RoboDK station: kr30 cnc 072119 second half.rdk

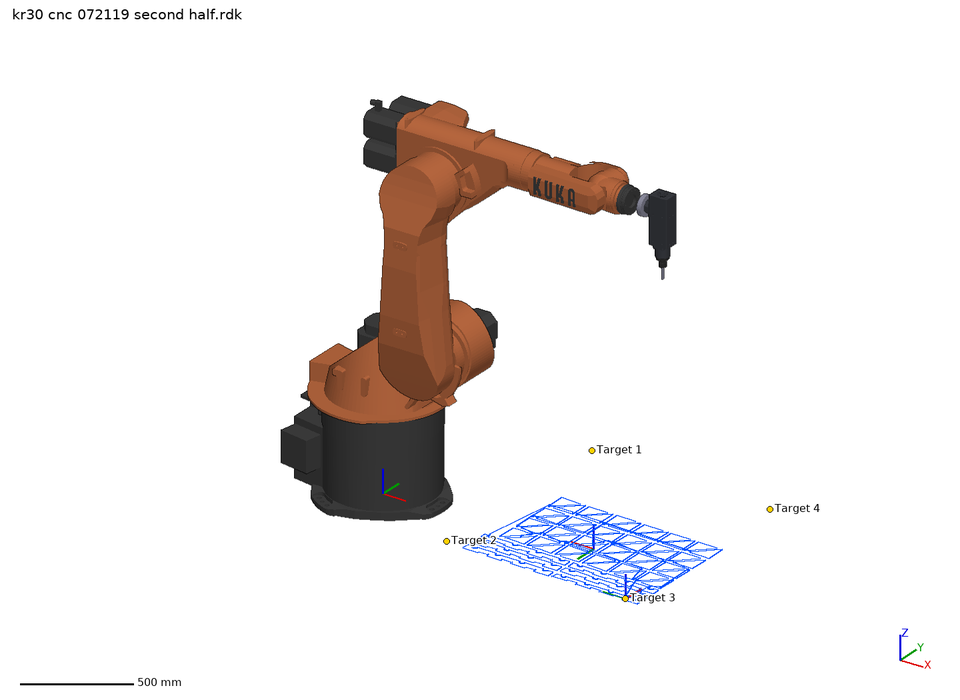
[picture v0: the station drawn from its stored meshes, robots at their saved joint values, targets as dots, program paths as lines]
Station kr30 cnc 072119 second half. Poses are relative to the parent item; angles as X-Y-Z fixed-axis rotations.
  - frame GIGASHEEN Base at (0, 0, 0) mm
    - robot GIGASHEEN (model KUKA KR 30 HA): 6 axes, payload 30 kg, reach 2033 mm, repeatability 0.05 mm, weight 665 kg
        modified DH rows (alpha deg, a mm, theta deg, d mm): 0, 0, 0, 815; -90, 350, 0, 0; 0, 850, -90, 0; -90, 145, 0, 820; 90, 0, 0, 0; -90, 0, 180, 170
        joint limits [-185, -135, -120, -350, -119, -350] to [185, 35, 158, 350, 119, 350]; home [0, -90, 90, 0, 0, 0]; saved at [0, -90, 90, 0, 0, 0]
      - tool 1/2" End Mill TCP, TCP at (337.71, -2.2, 160.57) mm, rotated rx 0 ry 90 rz 0 deg, size 415.8 x 102 x 153.6 mm
    - target Target 1 (joint target) at (982.46, 202.21, 406.25) mm, rotated rx -179.95 ry 0.15 rz -89.48 deg; joints [7.49, -59.642, 144.935, 97.969, -90.801, -4.608] of GIGASHEEN
    - target Target 2 (joint target) at (986.83, -921.64, 412.07) mm, rotated rx -179.94 ry 0.15 rz -89.48 deg; joints [51.766, -38.608, 94.384, 136.851, -116.554, -22.567] of GIGASHEEN
    - target Target 3 (joint target) at (1949.02, -919.97, 396.91) mm, rotated rx -179.94 ry 0.14 rz 179.61 deg; joints [29.5, -22.76, 62.288, 41.088, -47.759, -30.404] of GIGASHEEN
    - target Target 4 (joint target) at (1949.02, 190.94, 391.63) mm, rotated rx -179.94 ry 0.14 rz 179.61 deg; joints [-6.898, -35.989, 90.741, -8.88, -55.221, 5.167] of GIGASHEEN
  - machining project Machining Settings: C:/Users/liqui/OneDrive/Desktop/second half pipe jig.apt | rotZ(0) | rotX(0)*rotY(0) | rotZ(0)
  - program Prog2 (4 instructions, listed below)
  - frame Table at (1949.02, -919.97, 396.91) mm, rotated rx 0.87 ry 0.27 rz 90 deg
    - frame Frame 4 at (440, 480, -70) mm, rotated rx 0 ry 0 rz 90 deg
  - program Machining (1046 instructions, listed below)
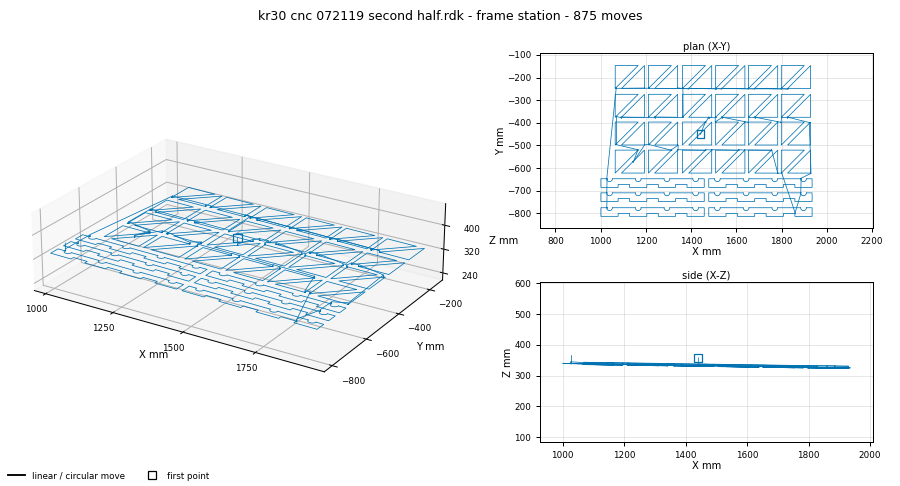
[picture p0: tool path of kr30 cnc 072119 second half.rdk in frame station, 875 of 879 moves have a stored position in this frame; points joined in program order, loops and branches not executed]

--- program Prog2 (robot GIGASHEEN) ---
  MoveJ (plywood back right safe) [its target is no longer in the station]
  MoveL (plywood back left safe) [its target is no longer in the station]
  MoveL (plywood front left safe) [its target is no longer in the station]
  MoveL (plywood front right safe) [its target is no longer in the station]

--- program Machining (robot GIGASHEEN) ---
  Smooth(1)
  Set Ref.: Frame 4
  Set Tool: 1/2" End Mill TCP
  Show 1/2" End Mill TCP
  Print: /'1001'
  Print: /''
  Print: /'2D Contour8'
  Set speed (500.0 mm/s)
  MoveJ 1 to (26.81, -31, 25) mm, rotated rx 180 ry 0 rz 0 deg; joints [21.751, -50.614, 128.61, 22.256, -77.995, -4.246]
  MoveL 2 to (26.81, -31, 25) mm, rotated rx 180 ry 0 rz 0 deg; joints [21.751, -50.614, 128.61, 22.256, -77.995, -4.246]
  MoveL 3 to (26.81, -31, 15) mm, rotated rx -180 ry 0 rz 0 deg; joints [21.756, -49.905, 128.509, 22.213, -78.558, -4.012]
  MoveL 4 to (26.81, -31, 15) mm, rotated rx -180 ry 0 rz 0 deg; joints [21.756, -49.905, 128.509, 22.213, -78.558, -4.012]
  Set speed (500.0 mm/s)
  MoveL 5 to (26.81, -31, 5) mm, rotated rx -180 ry 0 rz 0 deg; joints [21.761, -49.194, 128.4, 22.173, -79.115, -3.781]
  Set speed (25.4 mm/s)
  MoveL 6 to (26.81, -31, 1) mm, rotated rx -180 ry 0 rz 0 deg; joints [21.762, -48.909, 128.353, 22.158, -79.337, -3.69]
  MoveL 7 to (26.81, -31, -0.37) mm, rotated rx -180 ry 0 rz 0 deg; joints [21.763, -48.811, 128.337, 22.153, -79.412, -3.659]
  MoveC 8 to (26.94, -31.13, -0.81) mm, rotated rx -180 ry 0 rz 0 deg; joints [21.76, -48.784, 128.345, 22.147, -79.444, -3.645] to (27.26, -31.45, -1) mm, rotated rx 180 ry 0 rz 0 deg; joints [21.751, -48.782, 128.375, 22.136, -79.474, -3.631]
  Set speed (50.8 mm/s)
  MoveL 9 to (27.71, -31.9, -1) mm, rotated rx -180 ry 0 rz 0 deg; joints [21.739, -48.798, 128.421, 22.122, -79.5, -3.618]
  MoveC 10 to (27.89, -32.35, -1) mm, rotated rx -180 ry 0 rz 0 deg; joints [21.723, -48.807, 128.447, 22.104, -79.515, -3.608] to (27.71, -32.8, -1) mm, rotated rx -180 ry 0 rz 0 deg; joints [21.7, -48.806, 128.447, 22.081, -79.514, -3.604]
  MoveL 11 to (-23.07, -83.55, -1) mm, rotated rx 180 ry 0 rz 0 deg; joints [18.628, -47.91, 126.057, 19.06, -77.908, -3.574]
  MoveL 12 to (-23.07, 17.99, -1) mm, rotated rx 180 ry 0 rz 0 deg; joints [22.986, -46.905, 123.177, 23.67, -76.514, -5.195]
  MoveL 13 to (78.53, 17.99, -1) mm, rotated rx -180 ry 0 rz 0 deg; joints [24.923, -49.575, 130.527, 25.253, -80.933, -3.575]
  MoveL 14 to (27.71, -32.8, -1) mm, rotated rx -180 ry 0 rz 0 deg; joints [21.7, -48.806, 128.447, 22.081, -79.514, -3.604]
  MoveC 15 to (27.26, -32.98, -1) mm, rotated rx -180 ry 0 rz 0 deg; joints [21.683, -48.796, 128.419, 22.065, -79.497, -3.608] to (26.81, -32.8, -1) mm, rotated rx -180 ry 0 rz 0 deg; joints [21.684, -48.783, 128.381, 22.067, -79.474, -3.618]
  MoveL 16 to (26.36, -32.35, -1) mm, rotated rx -180 ry 0 rz 0 deg; joints [21.696, -48.767, 128.335, 22.082, -79.447, -3.631]
  MoveC 17 to (26.04, -32.03, -0.81) mm, rotated rx -180 ry 0 rz 0 deg; joints [21.704, -48.769, 128.305, 22.092, -79.418, -3.645] to (25.91, -31.9, -0.37) mm, rotated rx -180 ry 0 rz 0 deg; joints [21.707, -48.796, 128.297, 22.098, -79.385, -3.659]
  Set speed (500.0 mm/s)
  MoveL 18 to (25.91, -31.9, 5) mm, rotated rx -180 ry 0 rz 0 deg; joints [21.705, -49.179, 128.36, 22.119, -79.089, -3.781]
  MoveL 19 to (4.1, -85.45, 5) mm, rotated rx 180 ry 0 rz 0 deg; joints [18.952, -49.087, 128.208, 19.324, -78.85, -3.309]
  Set speed (25.4 mm/s)
  MoveL 20 to (4.1, -85.45, 1) mm, rotated rx -180 ry 0 rz 0 deg; joints [18.954, -48.802, 128.162, 19.311, -79.074, -3.229]
  MoveL 21 to (4.1, -85.45, -0.37) mm, rotated rx -180 ry 0 rz 0 deg; joints [18.954, -48.705, 128.146, 19.306, -79.151, -3.202]
  MoveC 22 to (4.1, -85.27, -0.81) mm, rotated rx -180 ry 0 rz 0 deg; joints [18.963, -48.672, 128.135, 19.314, -79.173, -3.195] to (4.1, -84.82, -1) mm, rotated rx 180 ry 0 rz 0 deg; joints [18.983, -48.655, 128.122, 19.334, -79.178, -3.198]
  Set speed (50.8 mm/s)
  MoveL 23 to (4.1, -84.18, -1) mm, rotated rx 180 ry 0 rz 0 deg; joints [19.012, -48.649, 128.106, 19.364, -79.169, -3.206]
  MoveC 24 to (4.29, -83.73, -1) mm, rotated rx 180 ry 0 rz 0 deg; joints [19.035, -48.65, 128.108, 19.387, -79.172, -3.21] to (4.74, -83.55, -1) mm, rotated rx 180 ry 0 rz 0 deg; joints [19.05, -48.661, 128.137, 19.402, -79.19, -3.207]
  MoveL 25 to (106.34, -83.55, -1) mm, rotated rx -180 ry 0 rz 0 deg; joints [20.764, -51.132, 135.495, 20.883, -83.861, -1.734]
  MoveL 26 to (106.34, 17.99, -1) mm, rotated rx -180 ry 0 rz 0 deg; joints [25.508, -50.235, 132.469, 25.761, -82.126, -3.095]
  MoveL 27 to (4.74, -83.55, -1) mm, rotated rx 180 ry 0 rz 0 deg; joints [19.05, -48.661, 128.137, 19.402, -79.19, -3.207]
  MoveC 28 to (4.29, -83.73, -1) mm, rotated rx -180 ry 0 rz 0 deg; joints [19.035, -48.65, 128.108, 19.387, -79.172, -3.21] to (3.84, -83.55, -1) mm, rotated rx 180 ry 0 rz 0 deg; joints [19.036, -48.637, 128.07, 19.39, -79.149, -3.219]
  MoveL 29 to (3.39, -83.1, -1) mm, rotated rx 180 ry 0 rz 0 deg; joints [19.05, -48.621, 128.025, 19.405, -79.122, -3.231]
  MoveC 30 to (3.07, -82.78, -0.81) mm, rotated rx -180 ry 0 rz 0 deg; joints [19.059, -48.623, 127.996, 19.417, -79.093, -3.243] to (2.94, -82.65, -0.37) mm, rotated rx -180 ry 0 rz 0 deg; joints [19.062, -48.651, 127.988, 19.423, -79.06, -3.256]
  Set speed (500.0 mm/s)
  MoveL 31 to (2.94, -82.65, 5) mm, rotated rx 180 ry 0 rz 0 deg; joints [19.06, -49.031, 128.05, 19.441, -78.76, -3.363]
  MoveL 32 to (-7.94, -102.8, 5) mm, rotated rx -180 ry 0 rz 0 deg; joints [17.99, -48.905, 127.74, 18.364, -78.518, -3.226]
  Set speed (25.4 mm/s)
  MoveL 33 to (-7.94, -102.8, 1) mm, rotated rx -180 ry 0 rz 0 deg; joints [17.992, -48.623, 127.693, 18.351, -78.743, -3.15]
  MoveL 34 to (-7.94, -102.8, -0.37) mm, rotated rx -180 ry 0 rz 0 deg; joints [17.992, -48.526, 127.677, 18.346, -78.819, -3.124]
  MoveC 35 to (-7.94, -102.98, -0.81) mm, rotated rx -180 ry 0 rz 0 deg; joints [17.984, -48.496, 127.676, 18.336, -78.847, -3.114] to (-7.94, -103.43, -1) mm, rotated rx 180 ry 0 rz 0 deg; joints [17.964, -48.486, 127.685, 18.314, -78.863, -3.104]
  Set speed (50.8 mm/s)
  MoveL 36 to (-7.94, -104.07, -1) mm, rotated rx 180 ry 0 rz 0 deg; joints [17.935, -48.491, 127.7, 18.285, -78.871, -3.096]
  MoveC 37 to (-8.13, -104.52, -1) mm, rotated rx 180 ry 0 rz 0 deg; joints [17.912, -48.49, 127.697, 18.261, -78.868, -3.092] to (-8.57, -104.7, -1) mm, rotated rx -180 ry 0 rz 0 deg; joints [17.897, -48.479, 127.668, 18.247, -78.849, -3.095]
  MoveL 38 to (-23.07, -104.7, -1) mm, rotated rx -180 ry 0 rz 0 deg; joints [17.689, -48.086, 126.578, 18.079, -78.174, -3.278]
  MoveL 39 to (-23.07, -206.24, -1) mm, rotated rx -180 ry 0 rz 0 deg; joints [13.051, -48.78, 128.687, 13.281, -79.301, -2.035]
  MoveL 40 to (78.53, -104.7, -1) mm, rotated rx 180 ry 0 rz 0 deg; joints [19.258, -50.66, 134.059, 19.406, -82.901, -1.917]
  MoveL 41 to (-8.57, -104.7, -1) mm, rotated rx -180 ry 0 rz 0 deg; joints [17.897, -48.479, 127.668, 18.247, -78.849, -3.095]
  MoveC 42 to (-9.02, -104.52, -1) mm, rotated rx -180 ry 0 rz 0 deg; joints [17.899, -48.466, 127.63, 18.251, -78.826, -3.103] to (-9.21, -104.07, -1) mm, rotated rx -180 ry 0 rz 0 deg; joints [17.917, -48.457, 127.605, 18.27, -78.812, -3.112]
  MoveL 43 to (-9.21, -103.43, -1) mm, rotated rx -180 ry 0 rz 0 deg; joints [17.945, -48.452, 127.59, 18.299, -78.804, -3.12]
  MoveC 44 to (-9.21, -102.98, -0.81) mm, rotated rx -180 ry 0 rz 0 deg; joints [17.965, -48.462, 127.581, 18.321, -78.788, -3.13] to (-9.21, -102.8, -0.37) mm, rotated rx 180 ry 0 rz 0 deg; joints [17.974, -48.492, 127.582, 18.331, -78.76, -3.141]
  Set speed (500.0 mm/s)
  MoveL 45 to (-9.21, -102.8, 5) mm, rotated rx -180 ry 0 rz 0 deg; joints [17.971, -48.871, 127.644, 18.349, -78.46, -3.242]
  MoveL 46 to (-41.36, -102.91, 5) mm, rotated rx -180 ry 0 rz 0 deg; joints [17.509, -47.974, 125.216, 17.98, -76.975, -3.637]
  Set speed (25.4 mm/s)
  MoveL 47 to (-41.36, -102.91, 1) mm, rotated rx -180 ry 0 rz 0 deg; joints [17.511, -47.7, 125.171, 17.966, -77.192, -3.565]
  MoveL 48 to (-41.36, -102.91, -0.36) mm, rotated rx -180 ry 0 rz 0 deg; joints [17.511, -47.607, 125.155, 17.961, -77.266, -3.541]
  MoveC 49 to (-41.23, -103.04, -0.81) mm, rotated rx -180 ry 0 rz 0 deg; joints [17.507, -47.581, 125.163, 17.955, -77.298, -3.529] to (-40.91, -103.35, -1) mm, rotated rx -180 ry 0 rz 0 deg; joints [17.498, -47.58, 125.193, 17.943, -77.327, -3.517]
  Set speed (50.8 mm/s)
  MoveL 50 to (-40.46, -103.8, -1) mm, rotated rx -180 ry 0 rz 0 deg; joints [17.484, -47.596, 125.238, 17.927, -77.353, -3.505]
  MoveC 51 to (-40.27, -104.25, -1) mm, rotated rx 180 ry 0 rz 0 deg; joints [17.467, -47.605, 125.263, 17.909, -77.367, -3.497] to (-40.46, -104.7, -1) mm, rotated rx 180 ry 0 rz 0 deg; joints [17.445, -47.604, 125.259, 17.886, -77.364, -3.493]
  MoveL 52 to (-142.06, -206.24, -1) mm, rotated rx 180 ry 0 rz 0 deg; joints [11.879, -45.301, 119.342, 12.39, -73.524, -3.11]
  MoveL 53 to (-68.27, -206.24, -1) mm, rotated rx -180 ry 0 rz 0 deg; joints [12.58, -47.525, 125.203, 12.905, -77.109, -2.46]
  MoveL 54 to (-40.46, -206.24, -1) mm, rotated rx -180 ry 0 rz 0 deg; joints [12.866, -48.308, 127.356, 13.131, -78.458, -2.201]
  MoveL 55 to (-40.46, -104.7, -1) mm, rotated rx -180 ry 0 rz 0 deg; joints [17.445, -47.604, 125.259, 17.886, -77.364, -3.493]
  MoveC 56 to (-40.27, -104.25, -1) mm, rotated rx 180 ry 0 rz 0 deg; joints [17.467, -47.605, 125.262, 17.909, -77.367, -3.497] to (-39.82, -104.07, -1) mm, rotated rx -180 ry 0 rz 0 deg; joints [17.482, -47.616, 125.292, 17.922, -77.386, -3.494]
  MoveL 57 to (-39.19, -104.07, -1) mm, rotated rx -180 ry 0 rz 0 deg; joints [17.49, -47.634, 125.341, 17.929, -77.415, -3.486]
  MoveC 58 to (-38.74, -104.07, -0.81) mm, rotated rx -180 ry 0 rz 0 deg; joints [17.497, -47.659, 125.377, 17.935, -77.426, -3.484] to (-38.55, -104.07, -0.37) mm, rotated rx -180 ry 0 rz 0 deg; joints [17.499, -47.695, 125.396, 17.938, -77.41, -3.49]
  Set speed (500.0 mm/s)
  MoveL 59 to (-38.55, -104.07, 5) mm, rotated rx -180 ry 0 rz 0 deg; joints [17.497, -48.063, 125.458, 17.957, -77.119, -3.586]
  MoveL 60 to (-38.55, -84.18, 5) mm, rotated rx -180 ry 0 rz 0 deg; joints [18.37, -47.893, 124.97, 18.874, -76.879, -3.877]
  Set speed (25.4 mm/s)
  MoveL 61 to (-38.55, -84.18, 1) mm, rotated rx -180 ry 0 rz 0 deg; joints [18.371, -47.621, 124.925, 18.859, -77.094, -3.802]
  MoveL 62 to (-38.55, -84.18, -0.37) mm, rotated rx -180 ry 0 rz 0 deg; joints [18.372, -47.528, 124.909, 18.854, -77.167, -3.776]
  MoveC 63 to (-38.74, -84.18, -0.81) mm, rotated rx -180 ry 0 rz 0 deg; joints [18.369, -47.492, 124.89, 18.85, -77.183, -3.77] to (-39.19, -84.18, -1) mm, rotated rx -180 ry 0 rz 0 deg; joints [18.363, -47.466, 124.854, 18.844, -77.172, -3.772]
  Set speed (50.8 mm/s)
  MoveL 64 to (-39.82, -84.18, -1) mm, rotated rx 180 ry 0 rz 0 deg; joints [18.354, -47.448, 124.806, 18.837, -77.142, -3.781]
  MoveC 65 to (-40.27, -84, -1) mm, rotated rx 180 ry 0 rz 0 deg; joints [18.355, -47.434, 124.767, 18.84, -77.119, -3.789] to (-40.46, -83.55, -1) mm, rotated rx -180 ry 0 rz 0 deg; joints [18.372, -47.425, 124.741, 18.859, -77.105, -3.798]
  MoveL 66 to (-40.46, 17.99, -1) mm, rotated rx 180 ry 0 rz 0 deg; joints [22.683, -46.409, 121.876, 23.438, -75.747, -5.457]
  MoveL 67 to (-142.06, -83.55, -1) mm, rotated rx -180 ry 0 rz 0 deg; joints [17.007, -44.359, 116.799, 17.867, -72.365, -5.039]
  MoveL 68 to (-68.27, -83.55, -1) mm, rotated rx -180 ry 0 rz 0 deg; joints [17.978, -46.625, 122.612, 18.557, -75.817, -4.148]
  MoveL 69 to (-40.46, -83.55, -1) mm, rotated rx -180 ry 0 rz 0 deg; joints [18.372, -47.425, 124.741, 18.859, -77.105, -3.798]
  MoveC 70 to (-40.01, -83.73, -1) mm, rotated rx -180 ry 0 rz 0 deg; joints [18.371, -47.439, 124.78, 18.855, -77.128, -3.79] to (-39.82, -84.18, -1) mm, rotated rx 180 ry 0 rz 0 deg; joints [18.354, -47.448, 124.806, 18.837, -77.142, -3.781]
  MoveL 71 to (-39.82, -84.82, -1) mm, rotated rx -180 ry 0 rz 0 deg; joints [18.326, -47.454, 124.822, 18.808, -77.15, -3.771]
  MoveC 72 to (-39.82, -85.27, -0.81) mm, rotated rx -180 ry 0 rz 0 deg; joints [18.306, -47.471, 124.835, 18.788, -77.146, -3.768] to (-39.82, -85.45, -0.37) mm, rotated rx -180 ry 0 rz 0 deg; joints [18.298, -47.503, 124.845, 18.781, -77.124, -3.774]
  Set speed (500.0 mm/s)
  MoveL 73 to (-39.82, -85.45, 5) mm, rotated rx 180 ry 0 rz 0 deg; joints [18.296, -47.868, 124.906, 18.801, -76.836, -3.874]
  MoveL 74 to (-67.63, -102.8, 5) mm, rotated rx -180 ry 0 rz 0 deg; joints [17.156, -47.209, 123.197, 17.712, -75.755, -3.953]
  Set speed (25.4 mm/s)
  MoveL 75 to (-67.63, -102.8, 1) mm, rotated rx -180 ry 0 rz 0 deg; joints [17.158, -46.943, 123.152, 17.696, -75.967, -3.884]
  MoveL 76 to (-67.63, -102.8, -0.37) mm, rotated rx 180 ry 0 rz 0 deg; joints [17.158, -46.852, 123.136, 17.691, -76.038, -3.86]
  MoveC 77 to (-67.63, -102.98, -0.81) mm, rotated rx -180 ry 0 rz 0 deg; joints [17.15, -46.824, 123.136, 17.681, -76.064, -3.85] to (-67.63, -103.43, -1) mm, rotated rx 180 ry 0 rz 0 deg; joints [17.131, -46.815, 123.144, 17.66, -76.079, -3.84]
  Set speed (50.8 mm/s)
  MoveL 78 to (-67.63, -104.07, -1) mm, rotated rx -180 ry 0 rz 0 deg; joints [17.104, -46.82, 123.159, 17.631, -76.087, -3.83]
  MoveC 79 to (-67.82, -104.52, -1) mm, rotated rx -180 ry 0 rz 0 deg; joints [17.082, -46.819, 123.155, 17.609, -76.083, -3.826] to (-68.27, -104.7, -1) mm, rotated rx -180 ry 0 rz 0 deg; joints [17.068, -46.807, 123.125, 17.596, -76.064, -3.828]
  MoveL 80 to (-169.87, -104.7, -1) mm, rotated rx 180 ry 0 rz 0 deg; joints [15.816, -43.643, 115.044, 16.72, -71.263, -4.993]
  MoveL 81 to (-169.87, -206.24, -1) mm, rotated rx 180 ry 0 rz 0 deg; joints [11.634, -44.407, 117.072, 12.225, -72.164, -3.345]
  MoveL 82 to (-68.27, -104.7, -1) mm, rotated rx 180 ry 0 rz 0 deg; joints [17.068, -46.807, 123.125, 17.596, -76.064, -3.828]
  MoveC 83 to (-67.82, -104.52, -1) mm, rotated rx -180 ry 0 rz 0 deg; joints [17.082, -46.819, 123.155, 17.609, -76.083, -3.826] to (-67.37, -104.7, -1) mm, rotated rx -180 ry 0 rz 0 deg; joints [17.08, -46.833, 123.195, 17.605, -76.106, -3.818]
  MoveL 84 to (-66.92, -105.15, -1) mm, rotated rx -180 ry 0 rz 0 deg; joints [17.066, -46.85, 123.24, 17.589, -76.132, -3.806]
  MoveC 85 to (-66.61, -105.47, -0.81) mm, rotated rx 180 ry 0 rz 0 deg; joints [17.057, -46.874, 123.274, 17.578, -76.141, -3.8] to (-66.47, -105.6, -0.37) mm, rotated rx 180 ry 0 rz 0 deg; joints [17.052, -46.909, 123.292, 17.575, -76.125, -3.805]
  Set speed (500.0 mm/s)
  MoveL 86 to (-66.47, -105.6, 5) mm, rotated rx -180 ry 0 rz 0 deg; joints [17.05, -47.267, 123.353, 17.595, -75.841, -3.897]
  MoveL 87 to (-168.97, -85.34, 5) mm, rotated rx 180 ry 0 rz 0 deg; joints [16.603, -43.86, 114.722, 17.603, -70.823, -5.418]
  Set speed (25.4 mm/s)
  MoveL 88 to (-168.97, -85.34, 1) mm, rotated rx -180 ry 0 rz 0 deg; joints [16.605, -43.618, 114.68, 17.584, -71.014, -5.355]
  MoveL 89 to (-168.97, -85.34, -0.37) mm, rotated rx -180 ry 0 rz 0 deg; joints [16.605, -43.536, 114.665, 17.577, -71.078, -5.334]
  MoveC 90 to (-169.1, -85.21, -0.81) mm, rotated rx -180 ry 0 rz 0 deg; joints [16.609, -43.503, 114.646, 17.58, -71.092, -5.33] to (-169.42, -84.89, -1) mm, rotated rx 180 ry 0 rz 0 deg; joints [16.618, -43.478, 114.611, 17.591, -71.082, -5.337]
  Set speed (50.8 mm/s)
  MoveL 91 to (-169.87, -84.45, -1) mm, rotated rx 180 ry 0 rz 0 deg; joints [16.631, -43.459, 114.563, 17.607, -71.056, -5.35]
  MoveC 92 to (-170.06, -84, -1) mm, rotated rx -180 ry 0 rz 0 deg; joints [16.647, -43.449, 114.537, 17.625, -71.043, -5.36] to (-169.87, -83.55, -1) mm, rotated rx -180 ry 0 rz 0 deg; joints [16.667, -43.451, 114.541, 17.646, -71.047, -5.366]
  MoveL 93 to (-68.27, 17.99, -1) mm, rotated rx 180 ry 0 rz 0 deg; joints [22.213, -45.592, 119.768, 23.09, -74.512, -5.868]
  MoveL 94 to (-169.87, 17.99, -1) mm, rotated rx -180 ry 0 rz 0 deg; joints [20.644, -42.362, 111.747, 22.043, -69.901, -7.322]
  MoveL 95 to (-169.87, -83.55, -1) mm, rotated rx 180 ry 0 rz 0 deg; joints [16.667, -43.451, 114.541, 17.646, -71.047, -5.366]
  MoveC 96 to (-170.06, -84, -1) mm, rotated rx 180 ry 0 rz 0 deg; joints [16.647, -43.449, 114.537, 17.625, -71.043, -5.36] to (-170.51, -84.18, -1) mm, rotated rx -180 ry 0 rz 0 deg; joints [16.634, -43.436, 114.505, 17.614, -71.024, -5.362]
  MoveL 97 to (-171.14, -84.18, -1) mm, rotated rx -180 ry 0 rz 0 deg; joints [16.626, -43.415, 114.453, 17.609, -70.993, -5.37]
  MoveC 98 to (-171.59, -84.18, -0.81) mm, rotated rx 180 ry 0 rz 0 deg; joints [16.621, -43.411, 114.418, 17.606, -70.963, -5.378] to (-171.77, -84.18, -0.37) mm, rotated rx -180 ry 0 rz 0 deg; joints [16.618, -43.432, 114.407, 17.607, -70.933, -5.387]
  Set speed (500.0 mm/s)
  MoveL 99 to (-171.77, -84.18, 5) mm, rotated rx 180 ry 0 rz 0 deg; joints [16.616, -43.755, 114.465, 17.633, -70.679, -5.472]
  MoveL 100 to (-183.66, -82.83, 5) mm, rotated rx 180 ry 0 rz 0 deg; joints [16.529, -43.341, 113.453, 17.606, -70.102, -5.634]
  Set speed (25.4 mm/s)
  MoveL 101 to (-183.66, -82.83, 1) mm, rotated rx -180 ry 0 rz 0 deg; joints [16.531, -43.102, 113.411, 17.586, -70.289, -5.571]
  MoveL 102 to (-183.66, -82.83, -0.37) mm, rotated rx -180 ry 0 rz 0 deg; joints [16.531, -43.021, 113.397, 17.579, -70.353, -5.55]
  MoveC 103 to (-183.84, -82.83, -0.81) mm, rotated rx -180 ry 0 rz 0 deg; joints [16.529, -42.987, 113.376, 17.576, -70.365, -5.545] to (-184.29, -82.83, -1) mm, rotated rx 180 ry 0 rz 0 deg; joints [16.524, -42.961, 113.337, 17.571, -70.352, -5.548]
  Set speed (50.8 mm/s)
  MoveL 104 to (-184.93, -82.83, -1) mm, rotated rx -180 ry 0 rz 0 deg; joints [16.517, -42.94, 113.285, 17.567, -70.322, -5.555]
  MoveC 105 to (-185.38, -82.64, -1) mm, rotated rx -180 ry 0 rz 0 deg; joints [16.519, -42.923, 113.243, 17.572, -70.298, -5.564] to (-185.56, -82.19, -1) mm, rotated rx -180 ry 0 rz 0 deg; joints [16.534, -42.912, 113.217, 17.59, -70.285, -5.574]
  MoveL 106 to (-185.56, 17.99, -1) mm, rotated rx 180 ry 0 rz 0 deg; joints [20.42, -41.828, 110.46, 21.912, -69.172, -7.543]
  MoveL 107 to (-287.16, -83.55, -1) mm, rotated rx -180 ry 0 rz 0 deg; joints [15.367, -39.281, 104.548, 16.947, -65.344, -6.733]
  MoveL 108 to (-185.56, -83.55, -1) mm, rotated rx 180 ry 0 rz 0 deg; joints [16.481, -42.925, 113.25, 17.531, -70.299, -5.549]
  MoveL 109 to (-185.56, -82.19, -1) mm, rotated rx -180 ry 0 rz 0 deg; joints [16.534, -42.912, 113.217, 17.59, -70.285, -5.574]
  MoveC 110 to (-185.38, -81.74, -1) mm, rotated rx -180 ry 0 rz 0 deg; joints [16.554, -42.914, 113.221, 17.611, -70.289, -5.58] to (-184.93, -81.56, -1) mm, rotated rx -180 ry 0 rz 0 deg; joints [16.567, -42.928, 113.254, 17.622, -70.309, -5.578]
  MoveL 111 to (-184.29, -81.56, -1) mm, rotated rx 180 ry 0 rz 0 deg; joints [16.575, -42.949, 113.306, 17.627, -70.339, -5.571]
  MoveC 112 to (-183.84, -81.56, -0.81) mm, rotated rx -180 ry 0 rz 0 deg; joints [16.58, -42.975, 113.345, 17.631, -70.352, -5.568] to (-183.66, -81.56, -0.37) mm, rotated rx -180 ry 0 rz 0 deg; joints [16.582, -43.008, 113.366, 17.634, -70.34, -5.573]
  Set speed (500.0 mm/s)
  MoveL 113 to (-183.66, -81.56, 5) mm, rotated rx 180 ry 0 rz 0 deg; joints [16.58, -43.329, 113.422, 17.661, -70.089, -5.657]
  MoveL 114 to (-187.42, -103.86, 5) mm, rotated rx -180 ry 0 rz 0 deg; joints [15.649, -43.408, 113.642, 16.661, -70.13, -5.292]
  Set speed (25.4 mm/s)
  MoveL 115 to (-187.42, -103.86, 1) mm, rotated rx 180 ry 0 rz 0 deg; joints [15.65, -43.169, 113.6, 16.642, -70.319, -5.233]
  MoveL 116 to (-187.42, -103.86, -0.37) mm, rotated rx 180 ry 0 rz 0 deg; joints [15.65, -43.087, 113.585, 16.636, -70.383, -5.213]
  MoveC 117 to (-187.29, -103.99, -0.81) mm, rotated rx -180 ry 0 rz 0 deg; joints [15.647, -43.066, 113.594, 16.629, -70.412, -5.202] to (-186.97, -104.31, -1) mm, rotated rx 180 ry 0 rz 0 deg; joints [15.638, -43.068, 113.626, 16.616, -70.439, -5.19]
  Set speed (50.8 mm/s)
  MoveL 118 to (-186.52, -104.76, -1) mm, rotated rx -180 ry 0 rz 0 deg; joints [15.625, -43.087, 113.673, 16.6, -70.465, -5.177]
  MoveC 119 to (-186.33, -105.21, -1) mm, rotated rx 180 ry 0 rz 0 deg; joints [15.609, -43.098, 113.699, 16.581, -70.478, -5.167] to (-186.52, -105.66, -1) mm, rotated rx 180 ry 0 rz 0 deg; joints [15.589, -43.095, 113.694, 16.56, -70.473, -5.161]
  MoveL 120 to (-199.47, -118.61, -1) mm, rotated rx -180 ry 0 rz 0 deg; joints [14.931, -42.768, 112.909, 15.91, -69.972, -5.072]
  MoveL 121 to (-287.16, -206.24, -1) mm, rotated rx -180 ry 0 rz 0 deg; joints [10.703, -40.298, 107.062, 11.694, -66.325, -4.315]
  MoveL 122 to (-185.56, -206.24, -1) mm, rotated rx -180 ry 0 rz 0 deg; joints [11.501, -43.889, 115.775, 12.139, -71.394, -3.477]
  MoveL 123 to (-185.56, -104.7, -1) mm, rotated rx -180 ry 0 rz 0 deg; joints [15.638, -43.119, 113.751, 16.609, -70.51, -5.168]
  MoveL 124 to (-186.52, -105.66, -1) mm, rotated rx -180 ry 0 rz 0 deg; joints [15.589, -43.095, 113.694, 16.56, -70.473, -5.161]
  MoveC 125 to (-186.97, -105.85, -1) mm, rotated rx -180 ry 0 rz 0 deg; joints [15.576, -43.082, 113.661, 16.549, -70.454, -5.163] to (-187.42, -105.66, -1) mm, rotated rx -180 ry 0 rz 0 deg; joints [15.579, -43.065, 113.62, 16.554, -70.43, -5.171]
  MoveL 126 to (-187.87, -105.21, -1) mm, rotated rx -180 ry 0 rz 0 deg; joints [15.592, -43.046, 113.572, 16.571, -70.404, -5.184]
  MoveC 127 to (-188.18, -104.89, -0.81) mm, rotated rx 180 ry 0 rz 0 deg; joints [15.601, -43.043, 113.541, 16.583, -70.377, -5.196] to (-188.32, -104.76, -0.37) mm, rotated rx 180 ry 0 rz 0 deg; joints [15.605, -43.065, 113.531, 16.59, -70.348, -5.206]
  Set speed (500.0 mm/s)
  MoveL 128 to (-188.32, -104.76, 5) mm, rotated rx -180 ry 0 rz 0 deg; joints [15.603, -43.385, 113.588, 16.615, -70.096, -5.286]
  MoveL 129 to (-212.74, -102.8, 5) mm, rotated rx -180 ry 0 rz 0 deg; joints [15.412, -42.522, 111.502, 16.544, -68.904, -5.591]
  Set speed (25.4 mm/s)
  MoveL 130 to (-212.74, -102.8, 1) mm, rotated rx -180 ry 0 rz 0 deg; joints [15.414, -42.288, 111.46, 16.524, -69.088, -5.533]
  MoveL 131 to (-212.74, -102.8, -0.37) mm, rotated rx -180 ry 0 rz 0 deg; joints [15.414, -42.208, 111.445, 16.518, -69.151, -5.513]
  MoveC 132 to (-212.74, -102.98, -0.81) mm, rotated rx 180 ry 0 rz 0 deg; joints [15.407, -42.184, 111.445, 16.507, -69.173, -5.503] to (-212.74, -103.43, -1) mm, rotated rx -180 ry 0 rz 0 deg; joints [15.389, -42.177, 111.453, 16.487, -69.186, -5.492]
  Set speed (50.8 mm/s)
  MoveL 133 to (-212.74, -104.07, -1) mm, rotated rx 180 ry 0 rz 0 deg; joints [15.364, -42.183, 111.468, 16.459, -69.192, -5.48]
  MoveC 134 to (-212.92, -104.52, -1) mm, rotated rx -180 ry 0 rz 0 deg; joints [15.345, -42.18, 111.463, 16.439, -69.187, -5.474] to (-213.37, -104.7, -1) mm, rotated rx 180 ry 0 rz 0 deg; joints [15.333, -42.166, 111.429, 16.428, -69.167, -5.475]
  MoveL 135 to (-314.97, -104.7, -1) mm, rotated rx -180 ry 0 rz 0 deg; joints [14.31, -38.414, 102.551, 15.937, -64.132, -6.607]
  MoveL 136 to (-314.97, -206.24, -1) mm, rotated rx -180 ry 0 rz 0 deg; joints [10.504, -39.239, 104.569, 11.607, -64.904, -4.546]
  MoveL 137 to (-213.37, -104.7, -1) mm, rotated rx 180 ry 0 rz 0 deg; joints [15.333, -42.166, 111.429, 16.428, -69.167, -5.475]
  MoveC 138 to (-212.92, -104.52, -1) mm, rotated rx -180 ry 0 rz 0 deg; joints [15.345, -42.18, 111.463, 16.439, -69.187, -5.474] to (-212.47, -104.7, -1) mm, rotated rx -180 ry 0 rz 0 deg; joints [15.342, -42.197, 111.505, 16.434, -69.211, -5.466]
  MoveL 139 to (-212.03, -105.15, -1) mm, rotated rx -180 ry 0 rz 0 deg; joints [15.329, -42.217, 111.553, 16.417, -69.237, -5.452]
  MoveC 140 to (-211.71, -105.47, -0.81) mm, rotated rx 180 ry 0 rz 0 deg; joints [15.32, -42.242, 111.589, 16.406, -69.247, -5.446] to (-211.58, -105.6, -0.37) mm, rotated rx -180 ry 0 rz 0 deg; joints [15.316, -42.274, 111.608, 16.403, -69.234, -5.448]
  Set speed (500.0 mm/s)
  MoveL 141 to (-211.58, -105.6, 5) mm, rotated rx -180 ry 0 rz 0 deg; joints [15.314, -42.589, 111.664, 16.429, -68.986, -5.525]
  MoveL 142 to (-314.07, -85.34, 5) mm, rotated rx -180 ry 0 rz 0 deg; joints [15.029, -38.583, 102.236, 16.797, -63.757, -7.097]
  Set speed (25.4 mm/s)
  MoveL 143 to (-314.07, -85.34, 1) mm, rotated rx -180 ry 0 rz 0 deg; joints [15.03, -38.367, 102.195, 16.774, -63.924, -7.042]
  MoveL 144 to (-314.07, -85.34, -0.37) mm, rotated rx -180 ry 0 rz 0 deg; joints [15.03, -38.294, 102.181, 16.766, -63.981, -7.023]
  MoveC 145 to (-314.21, -85.21, -0.81) mm, rotated rx -180 ry 0 rz 0 deg; joints [15.034, -38.263, 102.161, 16.769, -63.992, -7.021] to (-314.52, -84.89, -1) mm, rotated rx -180 ry 0 rz 0 deg; joints [15.043, -38.237, 102.123, 16.78, -63.981, -7.029]
  Set speed (50.8 mm/s)
  MoveL 146 to (-314.97, -84.45, -1) mm, rotated rx 180 ry 0 rz 0 deg; joints [15.055, -38.215, 102.071, 16.798, -63.954, -7.044]
  MoveC 147 to (-315.16, -84, -1) mm, rotated rx 180 ry 0 rz 0 deg; joints [15.069, -38.203, 102.043, 16.816, -63.941, -7.056] to (-314.97, -83.55, -1) mm, rotated rx -180 ry 0 rz 0 deg; joints [15.088, -38.206, 102.049, 16.836, -63.946, -7.064]
  MoveL 148 to (-213.37, 17.99, -1) mm, rotated rx 180 ry 0 rz 0 deg; joints [20.035, -40.857, 108.143, 21.699, -67.868, -7.937]
  MoveL 149 to (-314.97, 17.99, -1) mm, rotated rx -180 ry 0 rz 0 deg; joints [18.74, -37.033, 99.245, 21.139, -62.943, -9.408]
  MoveL 150 to (-314.97, -83.55, -1) mm, rotated rx 180 ry 0 rz 0 deg; joints [15.088, -38.206, 102.049, 16.836, -63.946, -7.064]
  MoveC 151 to (-315.16, -84, -1) mm, rotated rx -180 ry 0 rz 0 deg; joints [15.069, -38.203, 102.043, 16.816, -63.941, -7.056] to (-315.61, -84.18, -1) mm, rotated rx -180 ry 0 rz 0 deg; joints [15.058, -38.188, 102.007, 16.806, -63.92, -7.058]
  MoveL 152 to (-316.24, -84.18, -1) mm, rotated rx -180 ry 0 rz 0 deg; joints [15.052, -38.163, 101.949, 16.804, -63.887, -7.065]
  MoveC 153 to (-316.69, -84.18, -0.81) mm, rotated rx 180 ry 0 rz 0 deg; joints [15.047, -38.155, 101.91, 16.804, -63.857, -7.073] to (-316.88, -84.18, -0.37) mm, rotated rx -180 ry 0 rz 0 deg; joints [15.045, -38.172, 101.898, 16.806, -63.829, -7.082]
  Set speed (500.0 mm/s)
  MoveL 154 to (-316.88, -84.18, 5) mm, rotated rx -180 ry 0 rz 0 deg; joints [15.044, -38.46, 101.953, 16.837, -63.606, -7.156]
  MoveL 155 to (-329.06, -82.83, 5) mm, rotated rx -180 ry 0 rz 0 deg; joints [14.974, -37.961, 100.806, 16.854, -62.977, -7.332]
  Set speed (25.4 mm/s)
  MoveL 156 to (-329.06, -82.83, 1) mm, rotated rx -180 ry 0 rz 0 deg; joints [14.975, -37.748, 100.765, 16.83, -63.142, -7.277]
  MoveL 157 to (-329.06, -82.83, -0.36) mm, rotated rx -180 ry 0 rz 0 deg; joints [14.976, -37.675, 100.751, 16.822, -63.198, -7.258]
  MoveC 158 to (-329.24, -82.83, -0.81) mm, rotated rx 180 ry 0 rz 0 deg; joints [14.974, -37.644, 100.729, 16.819, -63.207, -7.254] to (-329.69, -82.83, -1) mm, rotated rx 180 ry 0 rz 0 deg; joints [14.97, -37.616, 100.686, 16.816, -63.191, -7.257]
  Set speed (50.8 mm/s)
  MoveL 159 to (-330.33, -82.83, -1) mm, rotated rx -180 ry 0 rz 0 deg; joints [14.964, -37.59, 100.628, 16.814, -63.159, -7.265]
  MoveC 160 to (-330.78, -82.64, -1) mm, rotated rx -180 ry 0 rz 0 deg; joints [14.966, -37.57, 100.582, 16.821, -63.134, -7.275] to (-330.96, -82.19, -1) mm, rotated rx -180 ry 0 rz 0 deg; joints [14.98, -37.558, 100.554, 16.839, -63.121, -7.287]
  MoveL 161 to (-330.96, 17.99, -1) mm, rotated rx -180 ry 0 rz 0 deg; joints [18.55, -36.388, 97.774, 21.084, -62.14, -9.649]
  MoveL 162 to (-432.56, -83.55, -1) mm, rotated rx 180 ry 0 rz 0 deg; joints [14.008, -33.239, 90.78, 16.622, -57.759, -8.56]
  MoveL 163 to (-330.96, -83.55, -1) mm, rotated rx -180 ry 0 rz 0 deg; joints [14.931, -37.572, 100.587, 16.782, -63.133, -7.257]
  MoveL 164 to (-330.96, -82.19, -1) mm, rotated rx -180 ry 0 rz 0 deg; joints [14.98, -37.558, 100.554, 16.839, -63.121, -7.287]
  MoveC 165 to (-330.78, -81.74, -1) mm, rotated rx -180 ry 0 rz 0 deg; joints [14.999, -37.561, 100.56, 16.859, -63.126, -7.295] to (-330.33, -81.56, -1) mm, rotated rx -180 ry 0 rz 0 deg; joints [15.01, -37.577, 100.596, 16.868, -63.147, -7.293]
  MoveL 166 to (-329.69, -81.56, -1) mm, rotated rx -180 ry 0 rz 0 deg; joints [15.016, -37.603, 100.655, 16.87, -63.18, -7.286]
  MoveC 167 to (-329.24, -81.56, -0.81) mm, rotated rx -180 ry 0 rz 0 deg; joints [15.02, -37.631, 100.698, 16.873, -63.195, -7.283] to (-329.06, -81.56, -0.37) mm, rotated rx 180 ry 0 rz 0 deg; joints [15.022, -37.662, 100.72, 16.876, -63.186, -7.287]
  Set speed (500.0 mm/s)
  MoveL 168 to (-329.06, -81.56, 5) mm, rotated rx -180 ry 0 rz 0 deg; joints [15.02, -37.947, 100.775, 16.908, -62.966, -7.361]
  MoveL 169 to (-332.82, -103.86, 5) mm, rotated rx 180 ry 0 rz 0 deg; joints [14.172, -38.019, 100.962, 15.948, -62.966, -6.908]
  Set speed (25.4 mm/s)
  MoveL 170 to (-332.82, -103.86, 1) mm, rotated rx -180 ry 0 rz 0 deg; joints [14.174, -37.806, 100.921, 15.925, -63.132, -6.856]
  MoveL 171 to (-332.82, -103.86, -0.36) mm, rotated rx -180 ry 0 rz 0 deg; joints [14.174, -37.733, 100.906, 15.917, -63.188, -6.838]
  MoveC 172 to (-332.69, -103.99, -0.81) mm, rotated rx -180 ry 0 rz 0 deg; joints [14.171, -37.716, 100.917, 15.91, -63.215, -6.828] to (-332.37, -104.31, -1) mm, rotated rx 180 ry 0 rz 0 deg; joints [14.162, -37.722, 100.951, 15.896, -63.241, -6.815]
  Set speed (50.8 mm/s)
  MoveL 173 to (-331.92, -104.76, -1) mm, rotated rx -180 ry 0 rz 0 deg; joints [14.15, -37.744, 101.003, 15.879, -63.268, -6.8]
  MoveC 174 to (-331.73, -105.21, -1) mm, rotated rx -180 ry 0 rz 0 deg; joints [14.135, -37.756, 101.031, 15.86, -63.281, -6.788] to (-331.92, -105.66, -1) mm, rotated rx -180 ry 0 rz 0 deg; joints [14.117, -37.753, 101.024, 15.84, -63.276, -6.78]
  MoveL 175 to (-344.87, -118.61, -1) mm, rotated rx -180 ry 0 rz 0 deg; joints [13.528, -37.354, 100.118, 15.254, -62.716, -6.644]
  MoveL 176 to (-432.56, -206.24, -1) mm, rotated rx -180 ry 0 rz 0 deg; joints [9.736, -34.354, 93.376, 11.414, -58.651, -5.575]
  MoveL 177 to (-330.96, -206.24, -1) mm, rotated rx 180 ry 0 rz 0 deg; joints [10.392, -38.614, 103.112, 11.564, -64.078, -4.68]
  MoveL 178 to (-330.96, -104.7, -1) mm, rotated rx 180 ry 0 rz 0 deg; joints [14.161, -37.782, 101.09, 15.884, -63.317, -6.79]
  MoveL 179 to (-331.92, -105.66, -1) mm, rotated rx -180 ry 0 rz 0 deg; joints [14.117, -37.753, 101.024, 15.84, -63.276, -6.78]
  MoveC 180 to (-332.37, -105.85, -1) mm, rotated rx -180 ry 0 rz 0 deg; joints [14.106, -37.736, 100.987, 15.831, -63.254, -6.781] to (-332.82, -105.66, -1) mm, rotated rx -180 ry 0 rz 0 deg; joints [14.109, -37.717, 100.941, 15.838, -63.23, -6.791]
  MoveL 181 to (-333.27, -105.21, -1) mm, rotated rx -180 ry 0 rz 0 deg; joints [14.121, -37.694, 100.889, 15.855, -63.203, -6.806]
  MoveC 182 to (-333.58, -104.89, -0.81) mm, rotated rx 180 ry 0 rz 0 deg; joints [14.129, -37.689, 100.855, 15.869, -63.176, -6.819] to (-333.71, -104.76, -0.37) mm, rotated rx -180 ry 0 rz 0 deg; joints [14.133, -37.706, 100.844, 15.877, -63.15, -6.829]
  Set speed (500.0 mm/s)
  MoveL 183 to (-333.71, -104.76, 5) mm, rotated rx -180 ry 0 rz 0 deg; joints [14.131, -37.992, 100.9, 15.907, -62.928, -6.899]
  MoveL 184 to (-358.14, -102.8, 5) mm, rotated rx -180 ry 0 rz 0 deg; joints [13.981, -36.975, 98.578, 15.926, -61.654, -7.227]
  Set speed (25.4 mm/s)
  MoveL 185 to (-358.14, -102.8, 1) mm, rotated rx -180 ry 0 rz 0 deg; joints [13.982, -36.766, 98.537, 15.903, -61.816, -7.175]
  MoveL 186 to (-358.14, -102.8, -0.37) mm, rotated rx -180 ry 0 rz 0 deg; joints [13.983, -36.694, 98.523, 15.895, -61.871, -7.158]
  MoveC 187 to (-358.14, -102.98, -0.81) mm, rotated rx -180 ry 0 rz 0 deg; joints [13.976, -36.672, 98.522, 15.885, -61.891, -7.148] to (-358.14, -103.43, -1) mm, rotated rx 180 ry 0 rz 0 deg; joints [13.96, -36.667, 98.531, 15.865, -61.902, -7.135]
  Set speed (50.8 mm/s)
  MoveL 188 to (-358.14, -104.07, -1) mm, rotated rx -180 ry 0 rz 0 deg; joints [13.937, -36.673, 98.546, 15.838, -61.908, -7.121]
  MoveC 189 to (-358.32, -104.52, -1) mm, rotated rx -180 ry 0 rz 0 deg; joints [13.919, -36.67, 98.539, 15.818, -61.902, -7.113] to (-358.77, -104.7, -1) mm, rotated rx -180 ry 0 rz 0 deg; joints [13.909, -36.653, 98.501, 15.809, -61.88, -7.114]
  MoveL 190 to (-460.37, -104.7, -1) mm, rotated rx -180 ry 0 rz 0 deg; joints [13.059, -32.178, 88.439, 15.736, -56.385, -8.392]
  MoveL 191 to (-460.37, -206.24, -1) mm, rotated rx 180 ry 0 rz 0 deg; joints [9.57, -33.089, 90.542, 11.415, -57.096, -5.84]
  MoveL 192 to (-358.77, -104.7, -1) mm, rotated rx -180 ry 0 rz 0 deg; joints [13.909, -36.653, 98.501, 15.809, -61.88, -7.114]
  MoveC 193 to (-358.32, -104.52, -1) mm, rotated rx -180 ry 0 rz 0 deg; joints [13.919, -36.67, 98.539, 15.818, -61.902, -7.113] to (-357.87, -104.7, -1) mm, rotated rx -180 ry 0 rz 0 deg; joints [13.917, -36.69, 98.585, 15.811, -61.927, -7.103]
  MoveL 194 to (-357.43, -105.15, -1) mm, rotated rx -180 ry 0 rz 0 deg; joints [13.905, -36.713, 98.638, 15.793, -61.954, -7.088]
  MoveC 195 to (-357.11, -105.47, -0.81) mm, rotated rx 180 ry 0 rz 0 deg; joints [13.896, -36.739, 98.677, 15.782, -61.965, -7.079] to (-356.98, -105.6, -0.37) mm, rotated rx 180 ry 0 rz 0 deg; joints [13.892, -36.769, 98.697, 15.779, -61.955, -7.08]
  Set speed (500.0 mm/s)
  MoveL 196 to (-356.98, -105.6, 5) mm, rotated rx -180 ry 0 rz 0 deg; joints [13.891, -37.051, 98.753, 15.81, -61.738, -7.149]
  MoveL 197 to (-455.42, -81.29, 5) mm, rotated rx -180 ry 0 rz 0 deg; joints [13.89, -32.45, 88.436, 16.774, -56.25, -9.019]
  Set speed (25.4 mm/s)
  MoveL 198 to (-455.42, -81.29, 1) mm, rotated rx -180 ry 0 rz 0 deg; joints [13.891, -32.255, 88.394, 16.746, -56.398, -8.967]
  MoveL 199 to (-455.42, -81.29, -0.37) mm, rotated rx -180 ry 0 rz 0 deg; joints [13.891, -32.188, 88.38, 16.736, -56.448, -8.949]
  MoveC 200 to (-455.55, -81.16, -0.81) mm, rotated rx -180 ry 0 rz 0 deg; joints [13.895, -32.158, 88.358, 16.739, -56.456, -8.948] to (-455.86, -80.84, -1) mm, rotated rx -180 ry 0 rz 0 deg; joints [13.903, -32.131, 88.315, 16.751, -56.442, -8.959]
  Set speed (50.8 mm/s)
  MoveL 201 to (-456.31, -80.39, -1) mm, rotated rx -180 ry 0 rz 0 deg; joints [13.914, -32.104, 88.256, 16.771, -56.413, -8.977]
  MoveC 202 to (-456.5, -79.94, -1) mm, rotated rx -180 ry 0 rz 0 deg; joints [13.928, -32.091, 88.225, 16.79, -56.399, -8.992] to (-456.31, -79.49, -1) mm, rotated rx 180 ry 0 rz 0 deg; joints [13.945, -32.094, 88.233, 16.809, -56.406, -9.001]
  MoveL 203 to (-358.77, 17.99, -1) mm, rotated rx 180 ry 0 rz 0 deg; joints [18.23, -35.235, 95.163, 21.009, -60.723, -10.078]
  MoveL 204 to (-460.37, 17.99, -1) mm, rotated rx 180 ry 0 rz 0 deg; joints [17.145, -30.647, 84.956, 21.013, -55.266, -11.804]
  MoveL 205 to (-460.37, -83.55, -1) mm, rotated rx -180 ry 0 rz 0 deg; joints [13.774, -31.948, 87.913, 16.64, -56.211, -8.952]
  MoveL 206 to (-456.31, -79.49, -1) mm, rotated rx -180 ry 0 rz 0 deg; joints [13.945, -32.094, 88.233, 16.809, -56.406, -9.001]
  MoveC 207 to (-455.86, -79.3, -1) mm, rotated rx -180 ry 0 rz 0 deg; joints [13.955, -32.113, 88.275, 16.817, -56.429, -9] to (-455.41, -79.49, -1) mm, rotated rx 180 ry 0 rz 0 deg; joints [13.952, -32.137, 88.327, 16.808, -56.456, -8.988]
  MoveL 208 to (-454.97, -79.94, -1) mm, rotated rx 180 ry 0 rz 0 deg; joints [13.941, -32.163, 88.385, 16.789, -56.485, -8.97]
  MoveC 209 to (-454.65, -80.26, -0.81) mm, rotated rx -180 ry 0 rz 0 deg; joints [13.933, -32.19, 88.428, 16.776, -56.499, -8.959] to (-454.52, -80.39, -0.37) mm, rotated rx -180 ry 0 rz 0 deg; joints [13.929, -32.22, 88.45, 16.774, -56.491, -8.96]
  Set speed (500.0 mm/s)
  MoveL 210 to (-454.52, -80.39, 5) mm, rotated rx -180 ry 0 rz 0 deg; joints [13.928, -32.482, 88.507, 16.811, -56.293, -9.03]
  MoveL 211 to (-462.28, 142.79, 5) mm, rotated rx -180 ry 0 rz 0 deg; joints [21.099, -28.744, 80.138, 26.572, -53.562, -15.937]
  Set speed (25.4 mm/s)
  MoveL 212 to (-462.28, 142.79, 1) mm, rotated rx 180 ry 0 rz 0 deg; joints [21.1, -28.557, 80.094, 26.526, -53.691, -15.858]
  MoveL 213 to (-462.28, 142.79, -0.36) mm, rotated rx -180 ry 0 rz 0 deg; joints [21.101, -28.493, 80.079, 26.511, -53.735, -15.832]
  MoveC 214 to (-462.09, 142.79, -0.81) mm, rotated rx -180 ry 0 rz 0 deg; joints [21.103, -28.482, 80.094, 26.505, -53.76, -15.818] to (-461.64, 142.79, -1) mm, rotated rx -180 ry 0 rz 0 deg; joints [21.109, -28.496, 80.142, 26.501, -53.791, -15.804]
  Set speed (50.8 mm/s)
  MoveL 215 to (-461.01, 142.79, -1) mm, rotated rx 180 ry 0 rz 0 deg; joints [21.116, -28.528, 80.212, 26.497, -53.827, -15.788]
  MoveC 216 to (-460.56, 142.61, -1) mm, rotated rx 180 ry 0 rz 0 deg; joints [21.116, -28.554, 80.269, 26.487, -53.855, -15.771] to (-460.37, 142.16, -1) mm, rotated rx 180 ry 0 rz 0 deg; joints [21.104, -28.572, 80.308, 26.466, -53.871, -15.751]
  MoveL 217 to (-460.37, 40.62, -1) mm, rotated rx -180 ry 0 rz 0 deg; joints [17.88, -30.31, 84.196, 21.996, -55.031, -12.482]
  MoveL 218 to (-358.77, 142.16, -1) mm, rotated rx -180 ry 0 rz 0 deg; joints [22.395, -33.33, 90.764, 26.29, -59.308, -13.522]
  MoveL 219 to (-460.37, 142.16, -1) mm, rotated rx 180 ry 0 rz 0 deg; joints [21.104, -28.572, 80.308, 26.466, -53.871, -15.751]
  MoveC 220 to (-460.82, 142.34, -1) mm, rotated rx 180 ry 0 rz 0 deg; joints [21.105, -28.546, 80.251, 26.476, -53.843, -15.768] to (-461.01, 142.79, -1) mm, rotated rx 180 ry 0 rz 0 deg; joints [21.116, -28.528, 80.212, 26.497, -53.827, -15.788]
  MoveL 221 to (-461.01, 143.43, -1) mm, rotated rx 180 ry 0 rz 0 deg; joints [21.136, -28.516, 80.185, 26.526, -53.819, -15.81]
  MoveC 222 to (-461.01, 143.88, -0.81) mm, rotated rx -180 ry 0 rz 0 deg; joints [21.15, -28.516, 80.168, 26.548, -53.808, -15.829] to (-461.01, 144.06, -0.37) mm, rotated rx -180 ry 0 rz 0 deg; joints [21.156, -28.533, 80.165, 26.561, -53.791, -15.844]
  Set speed (500.0 mm/s)
  MoveL 223 to (-461.01, 144.06, 5) mm, rotated rx -180 ry 0 rz 0 deg; joints [21.154, -28.785, 80.224, 26.622, -53.619, -15.95]
  MoveL 224 to (-417, 165.37, 5) mm, rotated rx 180 ry 0 rz 0 deg; joints [22.368, -30.545, 84.029, 27.395, -55.776, -15.62]
  Set speed (25.4 mm/s)
  MoveL 225 to (-417, 165.37, 1) mm, rotated rx -180 ry 0 rz 0 deg; joints [22.37, -30.355, 83.986, 27.35, -55.908, -15.538]
  MoveL 226 to (-417, 165.37, -0.37) mm, rotated rx 180 ry 0 rz 0 deg; joints [22.37, -30.29, 83.971, 27.335, -55.953, -15.511]
  MoveC 227 to (-417, 165.55, -0.81) mm, rotated rx -180 ry 0 rz 0 deg; joints [22.376, -30.264, 83.959, 27.338, -55.965, -15.508] to (-417, 166, -1) mm, rotated rx -180 ry 0 rz 0 deg; joints [22.39, -30.247, 83.937, 27.356, -55.966, -15.519]
  Set speed (50.8 mm/s)
  MoveL 228 to (-417, 166.64, -1) mm, rotated rx -180 ry 0 rz 0 deg; joints [22.41, -30.235, 83.91, 27.384, -55.958, -15.54]
  MoveC 229 to (-416.81, 167.09, -1) mm, rotated rx -180 ry 0 rz 0 deg; joints [22.427, -30.235, 83.91, 27.403, -55.962, -15.551] to (-416.36, 167.27, -1) mm, rotated rx 180 ry 0 rz 0 deg; joints [22.438, -30.253, 83.949, 27.41, -55.984, -15.546]
  MoveL 230 to (-314.76, 167.27, -1) mm, rotated rx -180 ry 0 rz 0 deg; joints [23.833, -34.756, 93.921, 27.452, -61.193, -13.398]
  MoveC 231 to (-302.06, 179.97, -1) mm, rotated rx -180 ry 0 rz 0 deg; joints [24.438, -35.052, 94.569, 28.031, -61.649, -13.521] to (-289.36, 167.27, -1) mm, rotated rx -180 ry 0 rz 0 deg; joints [24.207, -35.79, 96.247, 27.545, -62.427, -12.91]
  MoveL 232 to (-187.76, 167.27, -1) mm, rotated rx 180 ry 0 rz 0 deg; joints [25.822, -39.617, 105.023, 28.201, -67.145, -11.071]
  MoveC 233 to (-175.06, 179.97, -1) mm, rotated rx -180 ry 0 rz 0 deg; joints [26.482, -39.853, 105.557, 28.843, -67.537, -11.178] to (-162.36, 167.27, -1) mm, rotated rx -180 ry 0 rz 0 deg; joints [26.258, -40.504, 107.102, 28.431, -68.278, -10.629]
  MoveL 234 to (-60.76, 167.27, -1) mm, rotated rx -180 ry 0 rz 0 deg; joints [28.145, -43.803, 115.025, 29.607, -72.652, -8.879]
  MoveC 235 to (-48.06, 179.97, -1) mm, rotated rx 180 ry 0 rz 0 deg; joints [28.869, -43.989, 115.461, 30.317, -72.984, -8.959] to (-35.36, 167.27, -1) mm, rotated rx -180 ry 0 rz 0 deg; joints [28.656, -44.568, 116.918, 29.966, -73.71, -8.439]
  MoveL 236 to (-9.96, 167.27, -1) mm, rotated rx 180 ry 0 rz 0 deg; joints [29.184, -45.309, 118.777, 30.35, -74.754, -7.995]
  MoveL 237 to (-9.96, 205.37, -1) mm, rotated rx -180 ry 0 rz 0 deg; joints [30.608, -44.709, 117.196, 31.952, -74.131, -8.892]
  MoveL 238 to (-86.16, 205.37, -1) mm, rotated rx 180 ry 0 rz 0 deg; joints [29.026, -42.393, 111.534, 30.866, -71.003, -10.255]
  MoveL 239 to (-86.16, 192.67, -1) mm, rotated rx -180 ry 0 rz 0 deg; joints [28.571, -42.605, 112.065, 30.337, -71.197, -9.936]
  MoveL 240 to (-136.96, 192.67, -1) mm, rotated rx -180 ry 0 rz 0 deg; joints [27.607, -40.947, 108.108, 29.746, -69.028, -10.833]
  MoveL 241 to (-136.96, 205.37, -1) mm, rotated rx -180 ry 0 rz 0 deg; joints [28.052, -40.731, 107.577, 30.274, -68.843, -11.162]
  MoveL 242 to (-213.16, 205.37, -1) mm, rotated rx -180 ry 0 rz 0 deg; joints [26.699, -38.045, 101.332, 29.587, -65.474, -12.552]
  MoveL 243 to (-213.16, 192.67, -1) mm, rotated rx -180 ry 0 rz 0 deg; joints [26.269, -38.269, 101.866, 29.057, -65.649, -12.202]
  MoveL 244 to (-263.96, 192.67, -1) mm, rotated rx -180 ry 0 rz 0 deg; joints [25.443, -36.345, 97.472, 28.734, -63.301, -13.152]
  MoveL 245 to (-263.96, 205.37, -1) mm, rotated rx 180 ry 0 rz 0 deg; joints [25.863, -36.115, 96.933, 29.267, -63.131, -13.519]
  MoveL 246 to (-340.16, 205.37, -1) mm, rotated rx -180 ry 0 rz 0 deg; joints [24.696, -32.978, 89.911, 29.016, -59.443, -15.076]
  MoveL 247 to (-340.16, 192.67, -1) mm, rotated rx -180 ry 0 rz 0 deg; joints [24.29, -33.221, 90.464, 28.473, -59.609, -14.678]
  MoveL 248 to (-390.96, 192.67, -1) mm, rotated rx -180 ry 0 rz 0 deg; joints [23.574, -30.953, 85.457, 28.469, -57.009, -15.798]
  MoveL 249 to (-390.96, 205.37, -1) mm, rotated rx -180 ry 0 rz 0 deg; joints [23.972, -30.701, 84.889, 29.023, -56.844, -16.221]
  MoveL 250 to (-467.16, 205.37, -1) mm, rotated rx -180 ry 0 rz 0 deg; joints [22.957, -26.933, 76.699, 29.363, -52.678, -18.194]
  MoveL 251 to (-467.16, 167.27, -1) mm, rotated rx -180 ry 0 rz 0 deg; joints [21.798, -27.733, 78.463, 27.631, -53.173, -16.8]
  MoveL 252 to (-441.76, 167.27, -1) mm, rotated rx -180 ry 0 rz 0 deg; joints [22.114, -29.019, 81.255, 27.497, -54.599, -16.154]
  MoveC 253 to (-429.06, 179.97, -1) mm, rotated rx -180 ry 0 rz 0 deg; joints [22.67, -29.393, 82.057, 28.009, -55.135, -16.277] to (-416.36, 167.27, -1) mm, rotated rx 180 ry 0 rz 0 deg; joints [22.438, -30.253, 83.949, 27.41, -55.984, -15.546]
  MoveC 254 to (-416.55, 166.82, -1) mm, rotated rx 180 ry 0 rz 0 deg; joints [22.422, -30.253, 83.949, 27.391, -55.979, -15.536] to (-417, 166.64, -1) mm, rotated rx 180 ry 0 rz 0 deg; joints [22.41, -30.235, 83.91, 27.384, -55.958, -15.54]
  MoveL 255 to (-417.63, 166.64, -1) mm, rotated rx -180 ry 0 rz 0 deg; joints [22.402, -30.205, 83.844, 27.385, -55.923, -15.555]
  MoveC 256 to (-418.08, 166.64, -0.81) mm, rotated rx 180 ry 0 rz 0 deg; joints [22.396, -30.192, 83.799, 27.389, -55.893, -15.569] to (-418.27, 166.64, -0.37) mm, rotated rx -180 ry 0 rz 0 deg; joints [22.394, -30.205, 83.784, 27.394, -55.868, -15.582]
  Set speed (500.0 mm/s)
  MoveL 257 to (-418.27, 166.64, 5) mm, rotated rx -180 ry 0 rz 0 deg; joints [22.392, -30.46, 83.842, 27.454, -55.692, -15.692]
  MoveL 258 to (-417, 227.71, 5) mm, rotated rx -180 ry 0 rz 0 deg; joints [24.299, -29.277, 81.206, 30.156, -54.977, -17.775]
  Set speed (25.4 mm/s)
  MoveL 259 to (-417, 227.71, 1) mm, rotated rx 180 ry 0 rz 0 deg; joints [24.3, -29.089, 81.163, 30.107, -55.102, -17.687]
  MoveL 260 to (-417, 227.71, -0.37) mm, rotated rx 180 ry 0 rz 0 deg; joints [24.301, -29.025, 81.148, 30.09, -55.145, -17.658]
  MoveC 261 to (-417, 227.9, -0.81) mm, rotated rx -180 ry 0 rz 0 deg; joints [24.307, -28.999, 81.134, 30.093, -55.157, -17.654] to (-417, 228.34, -1) mm, rotated rx -180 ry 0 rz 0 deg; joints [24.32, -28.981, 81.11, 30.11, -55.156, -17.666]
  Set speed (50.8 mm/s)
  MoveL 262 to (-417, 228.98, -1) mm, rotated rx -180 ry 0 rz 0 deg; joints [24.34, -28.967, 81.08, 30.139, -55.148, -17.689]
  MoveC 263 to (-416.81, 229.43, -1) mm, rotated rx 180 ry 0 rz 0 deg; joints [24.356, -28.967, 81.078, 30.158, -55.152, -17.7] to (-416.36, 229.61, -1) mm, rotated rx -180 ry 0 rz 0 deg; joints [24.368, -28.985, 81.117, 30.164, -55.174, -17.695]
  MoveL 264 to (-314.76, 229.61, -1) mm, rotated rx 180 ry 0 rz 0 deg; joints [25.851, -33.589, 91.238, 30.098, -60.374, -15.295]
  MoveC 265 to (-302.06, 242.32, -1) mm, rotated rx -180 ry 0 rz 0 deg; joints [26.453, -33.867, 91.842, 30.671, -60.817, -15.424] to (-289.36, 229.62, -1) mm, rotated rx -180 ry 0 rz 0 deg; joints [26.248, -34.641, 93.587, 30.175, -61.6, -14.757]
  MoveL 266 to (-187.76, 229.61, -1) mm, rotated rx -180 ry 0 rz 0 deg; joints [27.957, -38.53, 102.414, 30.796, -66.271, -12.754]
  MoveC 267 to (-175.06, 242.31, -1) mm, rotated rx 180 ry 0 rz 0 deg; joints [28.613, -38.749, 102.9, 31.432, -66.648, -12.872] to (-162.36, 229.61, -1) mm, rotated rx 180 ry 0 rz 0 deg; joints [28.417, -39.43, 104.497, 31.024, -67.387, -12.278]
  MoveL 268 to (-60.76, 229.61, -1) mm, rotated rx -180 ry 0 rz 0 deg; joints [30.403, -42.776, 112.412, 32.206, -71.68, -10.417]
  MoveC 269 to (-48.06, 242.31, -1) mm, rotated rx 180 ry 0 rz 0 deg; joints [31.119, -42.945, 112.797, 32.908, -71.995, -10.514] to (-35.36, 229.61, -1) mm, rotated rx -180 ry 0 rz 0 deg; joints [30.939, -43.552, 114.296, 32.569, -72.713, -9.955]
  MoveL 270 to (-9.96, 229.61, -1) mm, rotated rx -180 ry 0 rz 0 deg; joints [31.492, -44.305, 116.146, 32.96, -73.731, -9.491]
  MoveL 271 to (-9.96, 267.71, -1) mm, rotated rx 180 ry 0 rz 0 deg; joints [32.849, -43.635, 114.426, 34.527, -73.099, -10.477]
  MoveL 272 to (-86.16, 267.71, -1) mm, rotated rx 180 ry 0 rz 0 deg; joints [31.201, -41.285, 108.782, 33.437, -70.04, -11.903]
  MoveL 273 to (-86.16, 255.01, -1) mm, rotated rx 180 ry 0 rz 0 deg; joints [30.766, -41.52, 109.362, 32.916, -70.238, -11.556]
  MoveL 274 to (-136.96, 255.01, -1) mm, rotated rx 180 ry 0 rz 0 deg; joints [29.756, -39.838, 105.406, 32.327, -68.108, -12.507]
  MoveL 275 to (-136.96, 267.71, -1) mm, rotated rx 180 ry 0 rz 0 deg; joints [30.182, -39.597, 104.826, 32.849, -67.917, -12.866]
  MoveL 276 to (-213.16, 267.71, -1) mm, rotated rx 180 ry 0 rz 0 deg; joints [28.763, -36.869, 98.559, 32.18, -64.592, -14.359]
  MoveL 277 to (-213.16, 255.01, -1) mm, rotated rx -180 ry 0 rz 0 deg; joints [28.349, -37.119, 99.145, 31.653, -64.775, -13.979]
  MoveL 278 to (-263.96, 255.01, -1) mm, rotated rx -180 ry 0 rz 0 deg; joints [27.478, -35.162, 94.722, 31.351, -62.449, -15.013]
  MoveL 279 to (-263.96, 267.71, -1) mm, rotated rx 180 ry 0 rz 0 deg; joints [27.883, -34.905, 94.128, 31.885, -62.271, -15.411]
  MoveL 280 to (-340.16, 267.71, -1) mm, rotated rx -180 ry 0 rz 0 deg; joints [26.653, -31.704, 87.023, 31.696, -58.601, -17.125]
  MoveL 281 to (-340.16, 255.01, -1) mm, rotated rx -180 ry 0 rz 0 deg; joints [26.259, -31.975, 87.635, 31.147, -58.776, -16.694]
  MoveL 282 to (-390.96, 255.01, -1) mm, rotated rx 180 ry 0 rz 0 deg; joints [25.502, -29.654, 82.546, 31.204, -56.179, -17.944]
  MoveL 283 to (-390.96, 267.71, -1) mm, rotated rx 180 ry 0 rz 0 deg; joints [25.887, -29.37, 81.914, 31.767, -56.004, -18.403]
  MoveL 284 to (-467.16, 267.71, -1) mm, rotated rx 180 ry 0 rz 0 deg; joints [24.812, -25.486, 73.523, 32.257, -51.818, -20.639]
  MoveL 285 to (-467.16, 229.61, -1) mm, rotated rx 180 ry 0 rz 0 deg; joints [23.685, -26.392, 75.508, 30.478, -52.351, -19.12]
  MoveL 286 to (-441.76, 229.61, -1) mm, rotated rx -180 ry 0 rz 0 deg; joints [24.022, -27.717, 78.367, 30.294, -53.784, -18.383]
  MoveC 287 to (-429.06, 242.31, -1) mm, rotated rx 180 ry 0 rz 0 deg; joints [24.578, -28.076, 79.132, 30.794, -54.312, -18.502] to (-416.36, 229.61, -1) mm, rotated rx -180 ry 0 rz 0 deg; joints [24.368, -28.985, 81.117, 30.164, -55.174, -17.695]
  MoveC 288 to (-416.55, 229.17, -1) mm, rotated rx -180 ry 0 rz 0 deg; joints [24.352, -28.985, 81.119, 30.145, -55.17, -17.684] to (-417, 228.98, -1) mm, rotated rx -180 ry 0 rz 0 deg; joints [24.34, -28.967, 81.08, 30.139, -55.148, -17.689]
  MoveL 289 to (-417.63, 228.98, -1) mm, rotated rx -180 ry 0 rz 0 deg; joints [24.331, -28.936, 81.012, 30.141, -55.114, -17.706]
  MoveC 290 to (-418.08, 228.98, -0.81) mm, rotated rx 180 ry 0 rz 0 deg; joints [24.325, -28.923, 80.967, 30.146, -55.084, -17.722] to (-418.27, 228.98, -0.37) mm, rotated rx -180 ry 0 rz 0 deg; joints [24.322, -28.935, 80.952, 30.152, -55.06, -17.736]
  Set speed (500.0 mm/s)
  MoveL 291 to (-418.27, 228.98, 5) mm, rotated rx -180 ry 0 rz 0 deg; joints [24.32, -29.187, 81.01, 30.218, -54.891, -17.854]
  MoveL 292 to (-391.6, 318.92, 5) mm, rotated rx -180 ry 0 rz 0 deg; joints [27.403, -28.406, 79.222, 34.143, -55.066, -20.5]
  Set speed (25.4 mm/s)
  MoveL 293 to (-391.6, 318.92, 1) mm, rotated rx -180 ry 0 rz 0 deg; joints [27.404, -28.219, 79.178, 34.089, -55.184, -20.403]
  MoveL 294 to (-391.6, 318.92, -0.36) mm, rotated rx -180 ry 0 rz 0 deg; joints [27.405, -28.156, 79.163, 34.071, -55.225, -20.37]
  MoveC 295 to (-391.6, 319.1, -0.81) mm, rotated rx 180 ry 0 rz 0 deg; joints [27.411, -28.13, 79.148, 34.073, -55.235, -20.367] to (-391.6, 319.55, -1) mm, rotated rx 180 ry 0 rz 0 deg; joints [27.424, -28.11, 79.121, 34.091, -55.234, -20.38]
  Set speed (50.8 mm/s)
  MoveL 296 to (-391.6, 320.19, -1) mm, rotated rx 180 ry 0 rz 0 deg; joints [27.443, -28.094, 79.086, 34.12, -55.225, -20.405]
  MoveC 297 to (-391.41, 320.64, -1) mm, rotated rx 180 ry 0 rz 0 deg; joints [27.459, -28.092, 79.081, 34.139, -55.228, -20.417] to (-390.96, 320.82, -1) mm, rotated rx 180 ry 0 rz 0 deg; joints [27.471, -28.11, 79.119, 34.145, -55.249, -20.411]
  MoveL 298 to (-340.16, 320.82, -1) mm, rotated rx 180 ry 0 rz 0 deg; joints [28.268, -30.502, 84.322, 34.003, -57.85, -19.007]
  MoveL 299 to (-340.16, 333.52, -1) mm, rotated rx 180 ry 0 rz 0 deg; joints [28.648, -30.197, 83.641, 34.559, -57.666, -19.477]
  MoveL 300 to (-263.96, 333.52, -1) mm, rotated rx -180 ry 0 rz 0 deg; joints [29.937, -33.481, 90.865, 34.657, -61.326, -17.579]
  MoveL 301 to (-263.96, 320.82, -1) mm, rotated rx -180 ry 0 rz 0 deg; joints [29.547, -33.768, 91.52, 34.121, -61.511, -17.146]
  MoveL 302 to (-213.16, 320.82, -1) mm, rotated rx 180 ry 0 rz 0 deg; joints [30.459, -35.766, 95.989, 34.385, -63.818, -16.018]
  MoveL 303 to (-213.16, 333.52, -1) mm, rotated rx 180 ry 0 rz 0 deg; joints [30.857, -35.488, 95.345, 34.912, -63.63, -16.432]
  MoveL 304 to (-136.96, 333.52, -1) mm, rotated rx -180 ry 0 rz 0 deg; joints [32.335, -38.268, 101.652, 35.541, -66.916, -14.825]
  MoveL 305 to (-136.96, 320.82, -1) mm, rotated rx 180 ry 0 rz 0 deg; joints [31.927, -38.536, 102.287, 35.023, -67.111, -14.433]
  MoveL 306 to (-86.16, 320.82, -1) mm, rotated rx 180 ry 0 rz 0 deg; joints [32.978, -40.246, 106.249, 35.599, -69.206, -13.423]
  MoveL 307 to (-86.16, 333.52, -1) mm, rotated rx 180 ry 0 rz 0 deg; joints [33.393, -39.985, 105.618, 36.113, -69.006, -13.803]
  MoveL 308 to (-9.96, 333.52, -1) mm, rotated rx 180 ry 0 rz 0 deg; joints [35.098, -42.375, 111.252, 37.188, -72.003, -12.31]
  MoveL 309 to (-9.96, 295.42, -1) mm, rotated rx -180 ry 0 rz 0 deg; joints [33.811, -43.12, 113.121, 35.654, -72.638, -11.228]
  MoveL 310 to (-35.36, 295.42, -1) mm, rotated rx 180 ry 0 rz 0 deg; joints [33.236, -42.355, 111.279, 35.264, -71.644, -11.712]
  MoveC 311 to (-48.06, 308.12, -1) mm, rotated rx 180 ry 0 rz 0 deg; joints [33.383, -41.716, 109.733, 35.594, -70.936, -12.314] to (-60.76, 295.42, -1) mm, rotated rx 180 ry 0 rz 0 deg; joints [32.678, -41.566, 109.4, 34.902, -70.634, -12.196]
  MoveL 312 to (-162.36, 295.42, -1) mm, rotated rx 180 ry 0 rz 0 deg; joints [30.605, -38.166, 101.478, 33.737, -66.416, -14.174]
  MoveC 313 to (-175.06, 308.12, -1) mm, rotated rx -180 ry 0 rz 0 deg; joints [30.772, -37.45, 99.822, 34.147, -65.678, -14.817] to (-187.76, 295.42, -1) mm, rotated rx -180 ry 0 rz 0 deg; joints [30.123, -37.25, 99.386, 33.519, -65.314, -14.686]
  MoveL 314 to (-289.36, 295.42, -1) mm, rotated rx 180 ry 0 rz 0 deg; joints [28.328, -33.284, 90.478, 32.961, -60.684, -16.874]
  MoveC 315 to (-302.06, 308.12, -1) mm, rotated rx 180 ry 0 rz 0 deg; joints [28.507, -32.467, 88.655, 33.473, -59.896, -17.603] to (-314.76, 295.42, -1) mm, rotated rx -180 ry 0 rz 0 deg; joints [27.909, -32.207, 88.096, 32.909, -59.463, -17.469]
  MoveL 316 to (-416.36, 295.42, -1) mm, rotated rx 180 ry 0 rz 0 deg; joints [26.343, -27.472, 77.768, 33.131, -54.26, -20.166]
  MoveC 317 to (-429.06, 308.12, -1) mm, rotated rx -180 ry 0 rz 0 deg; joints [26.53, -26.505, 75.669, 33.805, -53.382, -21.064] to (-441.76, 295.42, -1) mm, rotated rx -180 ry 0 rz 0 deg; joints [25.976, -26.16, 74.94, 33.319, -52.862, -20.95]
  MoveL 318 to (-467.16, 295.42, -1) mm, rotated rx -180 ry 0 rz 0 deg; joints [25.619, -24.783, 71.988, 33.573, -51.415, -21.798]
  MoveL 319 to (-467.16, 333.52, -1) mm, rotated rx -180 ry 0 rz 0 deg; joints [26.712, -23.75, 69.742, 35.419, -50.841, -23.474]
  MoveL 320 to (-390.96, 333.52, -1) mm, rotated rx 180 ry 0 rz 0 deg; joints [27.843, -27.79, 78.412, 34.721, -55.063, -20.914]
  MoveL 321 to (-390.96, 320.82, -1) mm, rotated rx 180 ry 0 rz 0 deg; joints [27.471, -28.11, 79.119, 34.145, -55.249, -20.411]
  MoveC 322 to (-391.15, 320.37, -1) mm, rotated rx 180 ry 0 rz 0 deg; joints [27.455, -28.112, 79.124, 34.126, -55.246, -20.399] to (-391.6, 320.19, -1) mm, rotated rx 180 ry 0 rz 0 deg; joints [27.443, -28.094, 79.086, 34.12, -55.225, -20.405]
  MoveL 323 to (-392.23, 320.19, -1) mm, rotated rx 180 ry 0 rz 0 deg; joints [27.433, -28.063, 79.019, 34.123, -55.192, -20.424]
  MoveC 324 to (-392.68, 320.19, -0.81) mm, rotated rx -180 ry 0 rz 0 deg; joints [27.426, -28.05, 78.973, 34.128, -55.162, -20.441] to (-392.87, 320.19, -0.37) mm, rotated rx -180 ry 0 rz 0 deg; joints [27.423, -28.062, 78.958, 34.134, -55.139, -20.458]
  Set speed (500.0 mm/s)
  MoveL 325 to (-392.87, 320.19, 5) mm, rotated rx -180 ry 0 rz 0 deg; joints [27.421, -28.311, 79.017, 34.207, -54.981, -20.587]
  MoveL 326 to (-332.82, 143, 5) mm, rotated rx -180 ry 0 rz 0 deg; joints [22.774, -34.728, 93.27, 26.431, -60.39, -13.162]
  Set speed (25.4 mm/s)
  MoveL 327 to (-332.82, 143, 1) mm, rotated rx 180 ry 0 rz 0 deg; joints [22.776, -34.526, 93.229, 26.392, -60.534, -13.08]
  MoveL 328 to (-332.82, 143, -0.36) mm, rotated rx 180 ry 0 rz 0 deg; joints [22.776, -34.458, 93.214, 26.379, -60.583, -13.053]
  MoveC 329 to (-332.69, 142.87, -0.81) mm, rotated rx -180 ry 0 rz 0 deg; joints [22.774, -34.443, 93.227, 26.37, -60.607, -13.037] to (-332.37, 142.55, -1) mm, rotated rx -180 ry 0 rz 0 deg; joints [22.768, -34.452, 93.268, 26.355, -60.634, -13.018]
  Set speed (50.8 mm/s)
  MoveL 330 to (-331.92, 142.1, -1) mm, rotated rx -180 ry 0 rz 0 deg; joints [22.759, -34.479, 93.327, 26.337, -60.662, -12.997]
  MoveC 331 to (-331.73, 141.65, -1) mm, rotated rx -180 ry 0 rz 0 deg; joints [22.747, -34.494, 93.363, 26.319, -60.676, -12.98] to (-331.92, 141.2, -1) mm, rotated rx 180 ry 0 rz 0 deg; joints [22.73, -34.494, 93.363, 26.299, -60.673, -12.971]
  MoveL 332 to (-344.87, 128.25, -1) mm, rotated rx -180 ry 0 rz 0 deg; joints [22.125, -34.165, 92.641, 25.72, -60.182, -12.844]
  MoveL 333 to (-432.56, 40.62, -1) mm, rotated rx 180 ry 0 rz 0 deg; joints [18.175, -31.639, 87.121, 21.938, -56.574, -11.952]
  MoveL 334 to (-330.96, 40.62, -1) mm, rotated rx 180 ry 0 rz 0 deg; joints [19.337, -36.083, 97.056, 22.041, -61.896, -10.22]
  MoveL 335 to (-330.96, 142.16, -1) mm, rotated rx 180 ry 0 rz 0 deg; joints [22.775, -34.518, 93.415, 26.342, -60.709, -12.98]
  MoveL 336 to (-331.92, 141.2, -1) mm, rotated rx -180 ry 0 rz 0 deg; joints [22.73, -34.494, 93.363, 26.299, -60.673, -12.971]
  MoveC 337 to (-332.37, 141.02, -1) mm, rotated rx -180 ry 0 rz 0 deg; joints [22.717, -34.478, 93.328, 26.29, -60.653, -12.974] to (-332.82, 141.2, -1) mm, rotated rx 180 ry 0 rz 0 deg; joints [22.717, -34.456, 93.278, 26.297, -60.628, -12.988]
  MoveL 338 to (-333.27, 141.65, -1) mm, rotated rx -180 ry 0 rz 0 deg; joints [22.726, -34.43, 93.218, 26.315, -60.6, -13.01]
  MoveC 339 to (-333.58, 141.97, -0.81) mm, rotated rx -180 ry 0 rz 0 deg; joints [22.732, -34.42, 93.178, 26.329, -60.574, -13.029] to (-333.71, 142.1, -0.37) mm, rotated rx -180 ry 0 rz 0 deg; joints [22.734, -34.435, 93.165, 26.339, -60.549, -13.044]
  Set speed (500.0 mm/s)
  MoveL 340 to (-333.71, 142.1, 5) mm, rotated rx -180 ry 0 rz 0 deg; joints [22.732, -34.705, 93.221, 26.391, -60.357, -13.153]
  MoveL 341 to (-316.88, 142.79, 5) mm, rotated rx -180 ry 0 rz 0 deg; joints [22.99, -35.398, 94.766, 26.466, -61.18, -12.854]
  Set speed (25.4 mm/s)
  MoveL 342 to (-316.88, 142.79, 1) mm, rotated rx 180 ry 0 rz 0 deg; joints [22.992, -35.194, 94.725, 26.428, -61.326, -12.772]
  MoveL 343 to (-316.88, 142.79, -0.36) mm, rotated rx -180 ry 0 rz 0 deg; joints [22.992, -35.125, 94.711, 26.415, -61.375, -12.745]
  MoveC 344 to (-316.69, 142.79, -0.81) mm, rotated rx -180 ry 0 rz 0 deg; joints [22.995, -35.109, 94.723, 26.412, -61.401, -12.732] to (-316.24, 142.79, -1) mm, rotated rx 180 ry 0 rz 0 deg; joints [23.002, -35.118, 94.763, 26.411, -61.429, -12.72]
  Set speed (50.8 mm/s)
  MoveL 345 to (-315.61, 142.79, -1) mm, rotated rx 180 ry 0 rz 0 deg; joints [23.011, -35.145, 94.822, 26.413, -61.461, -12.708]
  MoveC 346 to (-315.16, 142.61, -1) mm, rotated rx -180 ry 0 rz 0 deg; joints [23.011, -35.166, 94.87, 26.407, -61.485, -12.694] to (-314.97, 142.16, -1) mm, rotated rx -180 ry 0 rz 0 deg; joints [22.998, -35.181, 94.905, 26.389, -61.5, -12.678]
  MoveL 347 to (-314.97, 40.62, -1) mm, rotated rx 180 ry 0 rz 0 deg; joints [19.533, -36.731, 98.53, 22.096, -62.697, -9.968]
  MoveL 348 to (-301.06, 54.52, -1) mm, rotated rx -180 ry 0 rz 0 deg; joints [20.195, -37.092, 99.34, 22.739, -63.23, -10.098]
  MoveL 349 to (-213.37, 142.16, -1) mm, rotated rx 180 ry 0 rz 0 deg; joints [24.524, -39.105, 103.867, 26.944, -66.321, -10.868]
  MoveL 350 to (-314.97, 142.16, -1) mm, rotated rx -180 ry 0 rz 0 deg; joints [22.998, -35.181, 94.905, 26.389, -61.5, -12.678]
  MoveC 351 to (-315.42, 142.34, -1) mm, rotated rx -180 ry 0 rz 0 deg; joints [22.998, -35.16, 94.856, 26.395, -61.475, -12.692] to (-315.61, 142.79, -1) mm, rotated rx 180 ry 0 rz 0 deg; joints [23.011, -35.145, 94.822, 26.413, -61.461, -12.708]
  MoveL 352 to (-315.61, 143.43, -1) mm, rotated rx -180 ry 0 rz 0 deg; joints [23.032, -35.134, 94.797, 26.44, -61.453, -12.726]
  MoveC 353 to (-315.61, 143.88, -0.81) mm, rotated rx 180 ry 0 rz 0 deg; joints [23.047, -35.136, 94.781, 26.461, -61.44, -12.743] to (-315.61, 144.06, -0.37) mm, rotated rx -180 ry 0 rz 0 deg; joints [23.053, -35.155, 94.779, 26.473, -61.422, -12.757]
  Set speed (500.0 mm/s)
  MoveL 354 to (-315.61, 144.06, 5) mm, rotated rx 180 ry 0 rz 0 deg; joints [23.051, -35.429, 94.834, 26.524, -61.226, -12.867]
  MoveL 355 to (-287.8, 38.71, 5) mm, rotated rx -180 ry 0 rz 0 deg; joints [19.806, -38.149, 101.109, 22.176, -63.82, -9.609]
  Set speed (25.4 mm/s)
  MoveL 356 to (-287.8, 38.71, 1) mm, rotated rx 180 ry 0 rz 0 deg; joints [19.807, -37.936, 101.068, 22.146, -63.98, -9.538]
  MoveL 357 to (-287.8, 38.71, -0.37) mm, rotated rx 180 ry 0 rz 0 deg; joints [19.808, -37.863, 101.054, 22.135, -64.034, -9.513]
  MoveC 358 to (-287.8, 38.9, -0.81) mm, rotated rx 180 ry 0 rz 0 deg; joints [19.815, -37.836, 101.043, 22.14, -64.05, -9.51] to (-287.8, 39.35, -1) mm, rotated rx 180 ry 0 rz 0 deg; joints [19.831, -37.821, 101.027, 22.158, -64.052, -9.517]
  Set speed (50.8 mm/s)
  MoveL 359 to (-287.8, 39.98, -1) mm, rotated rx -180 ry 0 rz 0 deg; joints [19.853, -37.812, 101.007, 22.184, -64.045, -9.533]
  MoveC 360 to (-287.61, 40.43, -1) mm, rotated rx -180 ry 0 rz 0 deg; joints [19.871, -37.813, 101.009, 22.204, -64.049, -9.541] to (-287.16, 40.62, -1) mm, rotated rx -180 ry 0 rz 0 deg; joints [19.884, -37.828, 101.043, 22.214, -64.069, -9.539]
  MoveL 361 to (-185.56, 40.62, -1) mm, rotated rx -180 ry 0 rz 0 deg; joints [21.273, -41.545, 109.752, 22.878, -68.898, -8.027]
  MoveL 362 to (-185.56, 142.16, -1) mm, rotated rx -180 ry 0 rz 0 deg; joints [24.976, -40.099, 106.186, 27.169, -67.587, -10.395]
  MoveL 363 to (-287.16, 40.62, -1) mm, rotated rx 180 ry 0 rz 0 deg; joints [19.884, -37.828, 101.043, 22.214, -64.069, -9.539]
  MoveC 364 to (-287.61, 40.43, -1) mm, rotated rx 180 ry 0 rz 0 deg; joints [19.871, -37.813, 101.009, 22.204, -64.049, -9.541] to (-288.06, 40.62, -1) mm, rotated rx -180 ry 0 rz 0 deg; joints [19.872, -37.793, 100.963, 22.21, -64.025, -9.552]
  MoveL 365 to (-288.51, 41.07, -1) mm, rotated rx 180 ry 0 rz 0 deg; joints [19.882, -37.77, 100.908, 22.227, -63.998, -9.57]
  MoveC 366 to (-288.83, 41.38, -0.81) mm, rotated rx 180 ry 0 rz 0 deg; joints [19.89, -37.763, 100.871, 22.24, -63.971, -9.586] to (-288.96, 41.52, -0.37) mm, rotated rx 180 ry 0 rz 0 deg; joints [19.892, -37.78, 100.86, 22.249, -63.946, -9.599]
  Set speed (500.0 mm/s)
  MoveL 367 to (-288.96, 41.52, 5) mm, rotated rx 180 ry 0 rz 0 deg; joints [19.89, -38.066, 100.915, 22.289, -63.732, -9.696]
  MoveL 368 to (-168.01, 39.78, 5) mm, rotated rx -180 ry 0 rz 0 deg; joints [21.497, -42.505, 111.28, 23.031, -69.454, -7.871]
  Set speed (25.4 mm/s)
  MoveL 369 to (-168.01, 39.78, 1) mm, rotated rx -180 ry 0 rz 0 deg; joints [21.499, -42.272, 111.238, 23.005, -69.63, -7.792]
  MoveL 370 to (-168.01, 39.78, -0.36) mm, rotated rx -180 ry 0 rz 0 deg; joints [21.5, -42.192, 111.224, 22.996, -69.69, -7.765]
  MoveC 371 to (-168.15, 39.91, -0.81) mm, rotated rx 180 ry 0 rz 0 deg; joints [21.503, -42.16, 111.204, 22.998, -69.702, -7.761] to (-168.46, 40.23, -1) mm, rotated rx -180 ry 0 rz 0 deg; joints [21.51, -42.134, 111.166, 23.007, -69.692, -7.769]
  Set speed (50.8 mm/s)
  MoveL 372 to (-168.91, 40.68, -1) mm, rotated rx 180 ry 0 rz 0 deg; joints [21.52, -42.113, 111.115, 23.023, -69.666, -7.785]
  MoveC 373 to (-169.1, 41.13, -1) mm, rotated rx -180 ry 0 rz 0 deg; joints [21.535, -42.101, 111.086, 23.04, -69.652, -7.797] to (-168.91, 41.57, -1) mm, rotated rx -180 ry 0 rz 0 deg; joints [21.554, -42.102, 111.086, 23.061, -69.655, -7.804]
  MoveL 374 to (-68.27, 142.16, -1) mm, rotated rx -180 ry 0 rz 0 deg; joints [27.062, -43.955, 115.446, 28.447, -72.718, -8.426]
  MoveL 375 to (-169.87, 142.16, -1) mm, rotated rx 180 ry 0 rz 0 deg; joints [25.237, -40.646, 107.472, 27.309, -68.292, -10.13]
  MoveL 376 to (-169.87, 40.62, -1) mm, rotated rx -180 ry 0 rz 0 deg; joints [21.504, -42.082, 111.039, 23.012, -69.623, -7.798]
  MoveL 377 to (-168.91, 41.57, -1) mm, rotated rx -180 ry 0 rz 0 deg; joints [21.554, -42.102, 111.086, 23.061, -69.655, -7.804]
  MoveC 378 to (-168.46, 41.76, -1) mm, rotated rx -180 ry 0 rz 0 deg; joints [21.568, -42.115, 111.117, 23.073, -69.673, -7.801] to (-168.01, 41.57, -1) mm, rotated rx -180 ry 0 rz 0 deg; joints [21.568, -42.132, 111.16, 23.069, -69.696, -7.791]
  MoveL 379 to (-167.56, 41.13, -1) mm, rotated rx 180 ry 0 rz 0 deg; joints [21.557, -42.153, 111.211, 23.054, -69.722, -7.775]
  MoveC 380 to (-167.25, 40.81, -0.81) mm, rotated rx 180 ry 0 rz 0 deg; joints [21.55, -42.179, 111.249, 23.044, -69.732, -7.767] to (-167.12, 40.68, -0.37) mm, rotated rx 180 ry 0 rz 0 deg; joints [21.547, -42.211, 111.268, 23.043, -69.72, -7.771]
  Set speed (500.0 mm/s)
  MoveL 381 to (-167.12, 40.68, 5) mm, rotated rx -180 ry 0 rz 0 deg; joints [21.545, -42.525, 111.325, 23.078, -69.484, -7.878]
  MoveL 382 to (-142.69, 38.71, 5) mm, rotated rx 180 ry 0 rz 0 deg; joints [21.84, -43.369, 113.359, 23.219, -70.618, -7.482]
  Set speed (25.4 mm/s)
  MoveL 383 to (-142.69, 38.71, 1) mm, rotated rx 180 ry 0 rz 0 deg; joints [21.842, -43.131, 113.317, 23.194, -70.799, -7.4]
  MoveL 384 to (-142.69, 38.71, -0.37) mm, rotated rx -180 ry 0 rz 0 deg; joints [21.842, -43.049, 113.302, 23.185, -70.861, -7.373]
  MoveC 385 to (-142.69, 38.9, -0.81) mm, rotated rx -180 ry 0 rz 0 deg; joints [21.85, -43.02, 113.292, 23.191, -70.878, -7.367] to (-142.69, 39.35, -1) mm, rotated rx 180 ry 0 rz 0 deg; joints [21.867, -43.004, 113.275, 23.209, -70.881, -7.373]
  Set speed (50.8 mm/s)
  MoveL 386 to (-142.69, 39.98, -1) mm, rotated rx 180 ry 0 rz 0 deg; joints [21.891, -42.996, 113.255, 23.236, -70.873, -7.386]
  MoveC 387 to (-142.51, 40.43, -1) mm, rotated rx -180 ry 0 rz 0 deg; joints [21.911, -42.996, 113.255, 23.257, -70.876, -7.393] to (-142.06, 40.62, -1) mm, rotated rx 180 ry 0 rz 0 deg; joints [21.926, -43.008, 113.285, 23.269, -70.894, -7.39]
  MoveL 388 to (-40.46, 40.62, -1) mm, rotated rx 180 ry 0 rz 0 deg; joints [23.609, -46.146, 121.153, 24.437, -75.422, -5.872]
  MoveL 389 to (-40.46, 142.16, -1) mm, rotated rx -180 ry 0 rz 0 deg; joints [27.605, -44.794, 117.531, 28.829, -73.891, -7.956]
  MoveL 390 to (-142.06, 40.62, -1) mm, rotated rx -180 ry 0 rz 0 deg; joints [21.926, -43.008, 113.285, 23.269, -70.894, -7.39]
  MoveC 391 to (-142.51, 40.43, -1) mm, rotated rx -180 ry 0 rz 0 deg; joints [21.911, -42.996, 113.255, 23.257, -70.876, -7.393] to (-142.96, 40.62, -1) mm, rotated rx -180 ry 0 rz 0 deg; joints [21.912, -42.979, 113.213, 23.261, -70.853, -7.403]
  MoveL 392 to (-143.41, 41.07, -1) mm, rotated rx 180 ry 0 rz 0 deg; joints [21.922, -42.959, 113.163, 23.276, -70.827, -7.419]
  MoveC 393 to (-143.72, 41.38, -0.81) mm, rotated rx 180 ry 0 rz 0 deg; joints [21.929, -42.955, 113.13, 23.287, -70.8, -7.434] to (-143.85, 41.52, -0.37) mm, rotated rx -180 ry 0 rz 0 deg; joints [21.932, -42.976, 113.12, 23.294, -70.772, -7.448]
  Set speed (500.0 mm/s)
  MoveL 394 to (-143.85, 41.52, 5) mm, rotated rx 180 ry 0 rz 0 deg; joints [21.93, -43.295, 113.176, 23.329, -70.531, -7.557]
  MoveL 395 to (-22.17, 38.82, 5) mm, rotated rx 180 ry 0 rz 0 deg; joints [23.861, -47.088, 122.643, 24.638, -75.947, -5.698]
  Set speed (25.4 mm/s)
  MoveL 396 to (-22.17, 38.82, 1) mm, rotated rx -180 ry 0 rz 0 deg; joints [23.863, -46.824, 122.598, 24.617, -76.148, -5.604]
  MoveL 397 to (-22.17, 38.82, -0.36) mm, rotated rx -180 ry 0 rz 0 deg; joints [23.864, -46.733, 122.583, 24.61, -76.216, -5.572]
  MoveC 398 to (-22.31, 38.95, -0.81) mm, rotated rx 180 ry 0 rz 0 deg; joints [23.867, -46.698, 122.564, 24.612, -76.231, -5.566] to (-22.62, 39.27, -1) mm, rotated rx -180 ry 0 rz 0 deg; joints [23.874, -46.673, 122.528, 24.621, -76.221, -5.572]
  Set speed (50.8 mm/s)
  MoveL 399 to (-23.07, 39.72, -1) mm, rotated rx -180 ry 0 rz 0 deg; joints [23.885, -46.655, 122.48, 24.634, -76.195, -5.587]
  MoveC 400 to (-23.26, 40.17, -1) mm, rotated rx 180 ry 0 rz 0 deg; joints [23.9, -46.645, 122.451, 24.652, -76.18, -5.598] to (-23.07, 40.62, -1) mm, rotated rx 180 ry 0 rz 0 deg; joints [23.922, -46.645, 122.45, 24.674, -76.182, -5.604]
  MoveL 401 to (78.53, 142.16, -1) mm, rotated rx 180 ry 0 rz 0 deg; joints [30.172, -48.071, 126.033, 30.819, -78.747, -5.863]
  MoveL 402 to (60.76, 142.16, -1) mm, rotated rx -180 ry 0 rz 0 deg; joints [29.762, -47.614, 124.804, 30.483, -78.038, -6.187]
  MoveL 403 to (-23.07, 142.16, -1) mm, rotated rx -180 ry 0 rz 0 deg; joints [27.955, -45.305, 118.814, 29.083, -74.617, -7.659]
  MoveL 404 to (-23.07, 40.62, -1) mm, rotated rx -180 ry 0 rz 0 deg; joints [23.922, -46.645, 122.45, 24.674, -76.182, -5.604]
  MoveC 405 to (-23.26, 40.17, -1) mm, rotated rx -180 ry 0 rz 0 deg; joints [23.9, -46.645, 122.451, 24.652, -76.18, -5.598] to (-23.71, 39.98, -1) mm, rotated rx 180 ry 0 rz 0 deg; joints [23.884, -46.634, 122.424, 24.637, -76.163, -5.602]
  MoveL 406 to (-24.34, 39.98, -1) mm, rotated rx 180 ry 0 rz 0 deg; joints [23.872, -46.616, 122.377, 24.628, -76.136, -5.612]
  MoveC 407 to (-24.79, 39.98, -0.81) mm, rotated rx -180 ry 0 rz 0 deg; joints [23.864, -46.616, 122.346, 24.623, -76.107, -5.623] to (-24.98, 39.98, -0.37) mm, rotated rx 180 ry 0 rz 0 deg; joints [23.861, -46.64, 122.337, 24.623, -76.077, -5.636]
  Set speed (500.0 mm/s)
  MoveL 408 to (-24.98, 39.98, 5) mm, rotated rx 180 ry 0 rz 0 deg; joints [23.858, -46.994, 122.396, 24.651, -75.809, -5.762]
  MoveL 409 to (4.1, 38.71, 5) mm, rotated rx 180 ry 0 rz 0 deg; joints [24.344, -47.83, 124.583, 25.011, -77.083, -5.288]
  Set speed (25.4 mm/s)
  MoveL 410 to (4.1, 38.71, 1) mm, rotated rx -180 ry 0 rz 0 deg; joints [24.346, -47.559, 124.538, 24.992, -77.288, -5.191]
  MoveL 411 to (4.1, 38.71, -0.37) mm, rotated rx -180 ry 0 rz 0 deg; joints [24.347, -47.467, 124.522, 24.985, -77.358, -5.158]
  MoveC 412 to (4.1, 38.9, -0.81) mm, rotated rx 180 ry 0 rz 0 deg; joints [24.355, -47.434, 124.511, 24.991, -77.378, -5.15] to (4.1, 39.35, -1) mm, rotated rx -180 ry 0 rz 0 deg; joints [24.373, -47.416, 124.494, 25.01, -77.38, -5.154]
  Set speed (50.8 mm/s)
  MoveL 413 to (4.1, 39.98, -1) mm, rotated rx -180 ry 0 rz 0 deg; joints [24.4, -47.409, 124.473, 25.039, -77.371, -5.165]
  MoveC 414 to (4.29, 40.43, -1) mm, rotated rx -180 ry 0 rz 0 deg; joints [24.422, -47.409, 124.472, 25.062, -77.372, -5.17] to (4.74, 40.62, -1) mm, rotated rx -180 ry 0 rz 0 deg; joints [24.438, -47.419, 124.498, 25.077, -77.388, -5.166]
  MoveL 415 to (106.34, 40.62, -1) mm, rotated rx -180 ry 0 rz 0 deg; joints [26.518, -49.999, 131.709, 26.812, -81.72, -3.457]
  MoveL 416 to (106.34, 142.16, -1) mm, rotated rx -180 ry 0 rz 0 deg; joints [30.836, -48.764, 127.928, 31.373, -79.845, -5.345]
  MoveL 417 to (92.43, 128.25, -1) mm, rotated rx -180 ry 0 rz 0 deg; joints [29.934, -48.609, 127.535, 30.484, -79.552, -5.32]
  MoveL 418 to (4.74, 40.62, -1) mm, rotated rx -180 ry 0 rz 0 deg; joints [24.438, -47.419, 124.498, 25.077, -77.388, -5.166]
  MoveC 419 to (4.29, 40.43, -1) mm, rotated rx -180 ry 0 rz 0 deg; joints [24.422, -47.409, 124.471, 25.062, -77.372, -5.17] to (3.84, 40.62, -1) mm, rotated rx -180 ry 0 rz 0 deg; joints [24.421, -47.394, 124.433, 25.063, -77.349, -5.181]
  MoveL 420 to (3.39, 41.07, -1) mm, rotated rx 180 ry 0 rz 0 deg; joints [24.432, -47.377, 124.385, 25.076, -77.323, -5.196]
  MoveC 421 to (3.07, 41.38, -0.81) mm, rotated rx -180 ry 0 rz 0 deg; joints [24.439, -47.377, 124.353, 25.087, -77.295, -5.211] to (2.94, 41.52, -0.37) mm, rotated rx -180 ry 0 rz 0 deg; joints [24.442, -47.402, 124.345, 25.093, -77.264, -5.227]
  Set speed (500.0 mm/s)
  MoveL 422 to (2.94, 41.52, 5) mm, rotated rx -180 ry 0 rz 0 deg; joints [24.439, -47.765, 124.405, 25.119, -76.99, -5.358]
  MoveL 423 to (128.52, 38.82, 5) mm, rotated rx -180 ry 0 rz 0 deg; joints [26.932, -50.987, 133.366, 27.187, -82.341, -3.202]
  Set speed (25.4 mm/s)
  MoveL 424 to (128.52, 38.82, 1) mm, rotated rx 180 ry 0 rz 0 deg; joints [26.935, -50.68, 133.317, 27.174, -82.571, -3.084]
  MoveL 425 to (128.52, 38.82, -0.37) mm, rotated rx -180 ry 0 rz 0 deg; joints [26.935, -50.576, 133.3, 27.169, -82.649, -3.043]
  MoveC 426 to (128.39, 38.95, -0.81) mm, rotated rx -180 ry 0 rz 0 deg; joints [26.939, -50.537, 133.281, 27.171, -82.666, -3.035] to (128.07, 39.27, -1) mm, rotated rx -180 ry 0 rz 0 deg; joints [26.946, -50.512, 133.246, 27.179, -82.658, -3.04]
  Set speed (50.8 mm/s)
  MoveL 427 to (127.62, 39.72, -1) mm, rotated rx 180 ry 0 rz 0 deg; joints [26.956, -50.497, 133.2, 27.191, -82.63, -3.056]
  MoveC 428 to (127.44, 40.17, -1) mm, rotated rx -180 ry 0 rz 0 deg; joints [26.971, -50.489, 133.172, 27.208, -82.614, -3.066] to (127.62, 40.62, -1) mm, rotated rx -180 ry 0 rz 0 deg; joints [26.996, -50.488, 133.169, 27.233, -82.614, -3.07]
  MoveL 429 to (229.22, 142.16, -1) mm, rotated rx 180 ry 0 rz 0 deg; joints [34.108, -51.48, 135.919, 34.277, -84.529, -2.857]
  MoveL 430 to (187.76, 142.16, -1) mm, rotated rx 180 ry 0 rz 0 deg; joints [32.937, -50.628, 133.292, 33.21, -82.98, -3.738]
  MoveL 431 to (127.62, 142.16, -1) mm, rotated rx 180 ry 0 rz 0 deg; joints [31.361, -49.275, 129.357, 31.822, -80.676, -4.939]
  MoveL 432 to (127.62, 40.62, -1) mm, rotated rx -180 ry 0 rz 0 deg; joints [26.996, -50.488, 133.169, 27.233, -82.614, -3.07]
  MoveC 433 to (127.44, 40.17, -1) mm, rotated rx -180 ry 0 rz 0 deg; joints [26.971, -50.489, 133.172, 27.208, -82.614, -3.066] to (126.99, 39.98, -1) mm, rotated rx -180 ry 0 rz 0 deg; joints [26.953, -50.48, 133.147, 27.19, -82.599, -3.072]
  MoveL 434 to (126.35, 39.98, -1) mm, rotated rx 180 ry 0 rz 0 deg; joints [26.938, -50.466, 133.104, 27.178, -82.572, -3.083]
  MoveC 435 to (125.91, 39.98, -0.81) mm, rotated rx -180 ry 0 rz 0 deg; joints [26.928, -50.47, 133.076, 27.169, -82.543, -3.097] to (125.72, 39.98, -0.37) mm, rotated rx -180 ry 0 rz 0 deg; joints [26.924, -50.5, 133.069, 27.167, -82.51, -3.114]
  Set speed (500.0 mm/s)
  MoveL 436 to (125.72, 39.98, 5) mm, rotated rx 180 ry 0 rz 0 deg; joints [26.921, -50.91, 133.134, 27.185, -82.203, -3.272]
  MoveL 437 to (125.72, 18.63, 5) mm, rotated rx -180 ry 0 rz 0 deg; joints [25.956, -51.134, 133.858, 26.184, -82.593, -2.932]
  Set speed (25.4 mm/s)
  MoveL 438 to (125.72, 18.63, 1) mm, rotated rx -180 ry 0 rz 0 deg; joints [25.958, -50.825, 133.809, 26.171, -82.826, -2.816]
  MoveL 439 to (125.72, 18.63, -0.37) mm, rotated rx -180 ry 0 rz 0 deg; joints [25.959, -50.72, 133.792, 26.167, -82.906, -2.777]
  MoveC 440 to (125.91, 18.63, -0.81) mm, rotated rx -180 ry 0 rz 0 deg; joints [25.964, -50.689, 133.799, 26.169, -82.94, -2.761] to (126.35, 18.63, -1) mm, rotated rx 180 ry 0 rz 0 deg; joints [25.974, -50.685, 133.827, 26.178, -82.97, -2.747]
  Set speed (50.8 mm/s)
  MoveL 441 to (126.99, 18.63, -1) mm, rotated rx -180 ry 0 rz 0 deg; joints [25.988, -50.699, 133.871, 26.19, -82.997, -2.736]
  MoveC 442 to (127.44, 18.44, -1) mm, rotated rx -180 ry 0 rz 0 deg; joints [25.989, -50.711, 133.908, 26.191, -83.019, -2.725] to (127.62, 17.99, -1) mm, rotated rx 180 ry 0 rz 0 deg; joints [25.973, -50.719, 133.935, 26.173, -83.035, -2.715]
  MoveL 443 to (127.63, -83.55, -1) mm, rotated rx -180 ry 0 rz 0 deg; joints [21.162, -51.592, 136.992, 21.245, -84.842, -1.393]
  MoveL 444 to (229.22, 17.99, -1) mm, rotated rx -180 ry 0 rz 0 deg; joints [28.428, -52.756, 140.709, 28.453, -87.331, -0.703]
  MoveL 445 to (155.44, 17.99, -1) mm, rotated rx -180 ry 0 rz 0 deg; joints [26.605, -51.323, 135.826, 26.744, -84.218, -2.198]
  MoveL 446 to (127.62, 17.99, -1) mm, rotated rx -180 ry 0 rz 0 deg; joints [25.973, -50.719, 133.935, 26.173, -83.035, -2.715]
  MoveC 447 to (127.18, 18.18, -1) mm, rotated rx -180 ry 0 rz 0 deg; joints [25.971, -50.707, 133.898, 26.173, -83.013, -2.726] to (126.99, 18.63, -1) mm, rotated rx -180 ry 0 rz 0 deg; joints [25.988, -50.699, 133.871, 26.19, -82.997, -2.736]
  MoveL 448 to (126.99, 19.26, -1) mm, rotated rx 180 ry 0 rz 0 deg; joints [26.017, -50.693, 133.85, 26.22, -82.985, -2.746]
  MoveC 449 to (126.99, 19.71, -0.81) mm, rotated rx 180 ry 0 rz 0 deg; joints [26.037, -50.702, 133.837, 26.242, -82.966, -2.758] to (126.99, 19.9, -0.37) mm, rotated rx 180 ry 0 rz 0 deg; joints [26.045, -50.735, 133.837, 26.252, -82.936, -2.774]
  Set speed (500.0 mm/s)
  MoveL 450 to (126.99, 19.9, 5) mm, rotated rx -180 ry 0 rz 0 deg; joints [26.042, -51.15, 133.903, 26.269, -82.624, -2.929]
  MoveL 451 to (154.8, 38.71, 5) mm, rotated rx -180 ry 0 rz 0 deg; joints [27.539, -51.578, 135.149, 27.729, -83.434, -2.714]
  Set speed (25.4 mm/s)
  MoveL 452 to (154.8, 38.71, 1) mm, rotated rx -180 ry 0 rz 0 deg; joints [27.542, -51.263, 135.1, 27.718, -83.669, -2.59]
  MoveL 453 to (154.8, 38.71, -0.37) mm, rotated rx -180 ry 0 rz 0 deg; joints [27.542, -51.155, 135.082, 27.714, -83.749, -2.548]
  MoveC 454 to (154.8, 38.9, -0.81) mm, rotated rx -180 ry 0 rz 0 deg; joints [27.551, -51.118, 135.07, 27.721, -83.771, -2.537] to (154.8, 39.35, -1) mm, rotated rx -180 ry 0 rz 0 deg; joints [27.572, -51.099, 135.052, 27.742, -83.774, -2.539]
  Set speed (50.8 mm/s)
  MoveL 455 to (154.8, 39.98, -1) mm, rotated rx -180 ry 0 rz 0 deg; joints [27.601, -51.092, 135.03, 27.772, -83.761, -2.549]
  MoveC 456 to (154.99, 40.43, -1) mm, rotated rx -180 ry 0 rz 0 deg; joints [27.626, -51.091, 135.027, 27.797, -83.76, -2.552] to (155.44, 40.62, -1) mm, rotated rx 180 ry 0 rz 0 deg; joints [27.645, -51.099, 135.05, 27.815, -83.775, -2.546]
  MoveL 457 to (257.04, 40.62, -1) mm, rotated rx -180 ry 0 rz 0 deg; joints [30.279, -53.042, 141.682, 30.292, -87.956, -0.414]
  MoveL 458 to (257.04, 142.16, -1) mm, rotated rx -180 ry 0 rz 0 deg; joints [34.935, -52.013, 137.642, 35.047, -85.549, -2.237]
  MoveL 459 to (243.12, 128.25, -1) mm, rotated rx 180 ry 0 rz 0 deg; joints [33.911, -51.914, 137.368, 34.029, -85.36, -2.27]
  MoveL 460 to (155.44, 40.62, -1) mm, rotated rx 180 ry 0 rz 0 deg; joints [27.645, -51.099, 135.05, 27.815, -83.775, -2.546]
  MoveC 461 to (154.99, 40.43, -1) mm, rotated rx -180 ry 0 rz 0 deg; joints [27.626, -51.091, 135.027, 27.797, -83.76, -2.552] to (154.54, 40.62, -1) mm, rotated rx -180 ry 0 rz 0 deg; joints [27.623, -51.08, 134.99, 27.796, -83.738, -2.564]
  MoveL 462 to (154.09, 41.07, -1) mm, rotated rx -180 ry 0 rz 0 deg; joints [27.633, -51.066, 134.944, 27.807, -83.71, -2.58]
  MoveC 463 to (153.77, 41.38, -0.81) mm, rotated rx 180 ry 0 rz 0 deg; joints [27.64, -51.07, 134.914, 27.816, -83.68, -2.596] to (153.64, 41.52, -0.37) mm, rotated rx -180 ry 0 rz 0 deg; joints [27.642, -51.101, 134.906, 27.82, -83.646, -2.615]
  Set speed (500.0 mm/s)
  MoveL 464 to (153.64, 41.52, 5) mm, rotated rx -180 ry 0 rz 0 deg; joints [27.639, -51.523, 134.973, 27.836, -83.332, -2.781]
  MoveL 465 to (252.61, 16.27, 5) mm, rotated rx -180 ry 0 rz 0 deg; joints [28.965, -53.704, 142.361, 28.977, -87.955, -0.379]
  Set speed (25.4 mm/s)
  MoveL 466 to (252.61, 16.27, 1) mm, rotated rx -180 ry 0 rz 0 deg; joints [28.968, -53.348, 142.306, 28.975, -88.219, -0.232]
  MoveL 467 to (252.61, 16.27, -0.36) mm, rotated rx -180 ry 0 rz 0 deg; joints [28.968, -53.226, 142.287, 28.974, -88.309, -0.183]
  MoveC 468 to (252.74, 16.14, -0.81) mm, rotated rx -180 ry 0 rz 0 deg; joints [28.966, -53.189, 142.293, 28.971, -88.347, -0.162] to (253.06, 15.82, -1) mm, rotated rx 180 ry 0 rz 0 deg; joints [28.959, -53.18, 142.322, 28.964, -88.38, -0.143]
  Set speed (50.8 mm/s)
  MoveL 469 to (253.51, 15.37, -1) mm, rotated rx -180 ry 0 rz 0 deg; joints [28.949, -53.191, 142.367, 28.953, -88.409, -0.127]
  MoveC 470 to (253.7, 14.92, -1) mm, rotated rx -180 ry 0 rz 0 deg; joints [28.932, -53.198, 142.394, 28.936, -88.428, -0.116] to (253.51, 14.47, -1) mm, rotated rx 180 ry 0 rz 0 deg; joints [28.905, -53.198, 142.398, 28.909, -88.43, -0.114]
  MoveL 471 to (155.44, -83.55, -1) mm, rotated rx 180 ry 0 rz 0 deg; joints [21.703, -52.16, 138.925, 21.748, -86.125, -0.926]
  MoveL 472 to (229.23, -83.55, -1) mm, rotated rx -180 ry 0 rz 0 deg; joints [23.275, -53.471, 143.935, 23.269, -89.557, 0.456]
  MoveL 473 to (257.04, -83.55, -1) mm, rotated rx 180 ry 0 rz 0 deg; joints [23.925, -53.883, 145.779, 23.92, -90.863, 1.041]
  MoveL 474 to (257.04, 17.99, -1) mm, rotated rx -180 ry 0 rz 0 deg; joints [29.175, -53.228, 142.499, 29.178, -88.494, -0.083]
  MoveL 475 to (253.51, 14.47, -1) mm, rotated rx -180 ry 0 rz 0 deg; joints [28.905, -53.198, 142.398, 28.909, -88.43, -0.114]
  MoveC 476 to (253.06, 14.28, -1) mm, rotated rx -180 ry 0 rz 0 deg; joints [28.883, -53.192, 142.376, 28.888, -88.416, -0.122] to (252.61, 14.47, -1) mm, rotated rx 180 ry 0 rz 0 deg; joints [28.88, -53.183, 142.341, 28.885, -88.393, -0.135]
  MoveL 477 to (252.16, 14.92, -1) mm, rotated rx -180 ry 0 rz 0 deg; joints [28.89, -53.172, 142.296, 28.895, -88.363, -0.151]
  MoveC 478 to (251.85, 15.24, -0.81) mm, rotated rx -180 ry 0 rz 0 deg; joints [28.897, -53.181, 142.267, 28.903, -88.33, -0.169] to (251.71, 15.37, -0.37) mm, rotated rx 180 ry 0 rz 0 deg; joints [28.9, -53.218, 142.261, 28.906, -88.292, -0.191]
  Set speed (500.0 mm/s)
  MoveL 479 to (251.71, 15.37, 5) mm, rotated rx -180 ry 0 rz 0 deg; joints [28.896, -53.696, 142.335, 28.909, -87.938, -0.386]
  MoveL 480 to (272.52, 17.28, 5) mm, rotated rx -180 ry 0 rz 0 deg; joints [29.567, -54.026, 143.595, 29.567, -88.755, 0.059]
  Set speed (25.4 mm/s)
  MoveL 481 to (272.52, 17.28, 1) mm, rotated rx -180 ry 0 rz 0 deg; joints [29.57, -53.661, 143.539, 29.567, -89.024, 0.212]
  MoveL 482 to (272.52, 17.28, -0.36) mm, rotated rx -180 ry 0 rz 0 deg; joints [29.571, -53.537, 143.519, 29.567, -89.115, 0.264]
  MoveC 483 to (272.7, 17.28, -0.81) mm, rotated rx -180 ry 0 rz 0 deg; joints [29.577, -53.498, 143.524, 29.572, -89.153, 0.285] to (273.15, 17.28, -1) mm, rotated rx -180 ry 0 rz 0 deg; joints [29.589, -53.488, 143.55, 29.585, -89.184, 0.303]
  Set speed (50.8 mm/s)
  MoveL 484 to (273.79, 17.28, -1) mm, rotated rx -180 ry 0 rz 0 deg; joints [29.607, -53.498, 143.59, 29.603, -89.211, 0.318]
  MoveC 485 to (274.24, 17.09, -1) mm, rotated rx -180 ry 0 rz 0 deg; joints [29.611, -53.506, 143.625, 29.606, -89.234, 0.331] to (274.42, 16.64, -1) mm, rotated rx -180 ry 0 rz 0 deg; joints [29.594, -53.513, 143.653, 29.589, -89.253, 0.342]
  MoveL 486 to (274.42, -83.55, -1) mm, rotated rx -180 ry 0 rz 0 deg; joints [24.348, -54.116, 146.919, 24.353, -91.685, 1.428]
  MoveL 487 to (376.02, 17.99, -1) mm, rotated rx -180 ry 0 rz 0 deg; joints [32.82, -54.758, 149.844, 32.877, -93.404, 3.031]
  MoveL 488 to (274.42, 17.99, -1) mm, rotated rx -180 ry 0 rz 0 deg; joints [29.661, -53.502, 143.605, 29.656, -89.219, 0.323]
  MoveL 489 to (274.42, 16.64, -1) mm, rotated rx -180 ry 0 rz 0 deg; joints [29.594, -53.513, 143.653, 29.589, -89.253, 0.342]
  MoveC 490 to (274.24, 16.19, -1) mm, rotated rx 180 ry 0 rz 0 deg; joints [29.566, -53.513, 143.657, 29.561, -89.256, 0.343] to (273.79, 16.01, -1) mm, rotated rx -180 ry 0 rz 0 deg; joints [29.544, -53.508, 143.636, 29.539, -89.242, 0.335]
  MoveL 491 to (273.15, 16.01, -1) mm, rotated rx 180 ry 0 rz 0 deg; joints [29.526, -53.498, 143.595, 29.521, -89.215, 0.32]
  MoveC 492 to (272.7, 16.01, -0.81) mm, rotated rx -180 ry 0 rz 0 deg; joints [29.513, -53.508, 143.57, 29.509, -89.184, 0.303] to (272.52, 16.01, -0.37) mm, rotated rx 180 ry 0 rz 0 deg; joints [29.508, -53.546, 143.564, 29.503, -89.146, 0.281]
  Set speed (500.0 mm/s)
  MoveL 493 to (272.52, 16.01, 5) mm, rotated rx 180 ry 0 rz 0 deg; joints [29.504, -54.036, 143.64, 29.504, -88.786, 0.077]
  MoveL 494 to (324.31, 93.16, 5) mm, rotated rx -180 ry 0 rz 0 deg; joints [34.836, -54.188, 143.857, 34.835, -88.858, 0.083]
  Set speed (25.4 mm/s)
  MoveL 495 to (324.31, 93.16, 1) mm, rotated rx 180 ry 0 rz 0 deg; joints [34.839, -53.821, 143.801, 34.835, -89.113, 0.261]
  MoveL 496 to (324.31, 93.16, -0.36) mm, rotated rx -180 ry 0 rz 0 deg; joints [34.84, -53.696, 143.781, 34.835, -89.2, 0.321]
  MoveC 497 to (324.44, 93.03, -0.81) mm, rotated rx 180 ry 0 rz 0 deg; joints [34.838, -53.658, 143.788, 34.833, -89.237, 0.347] to (324.75, 92.71, -1) mm, rotated rx -180 ry 0 rz 0 deg; joints [34.834, -53.648, 143.817, 34.828, -89.269, 0.369]
  Set speed (50.8 mm/s)
  MoveL 498 to (325.2, 92.27, -1) mm, rotated rx 180 ry 0 rz 0 deg; joints [34.827, -53.659, 143.863, 34.821, -89.298, 0.389]
  MoveC 499 to (325.39, 91.82, -1) mm, rotated rx 180 ry 0 rz 0 deg; joints [34.812, -53.665, 143.892, 34.806, -89.317, 0.402] to (325.2, 91.37, -1) mm, rotated rx -180 ry 0 rz 0 deg; joints [34.785, -53.667, 143.9, 34.779, -89.322, 0.405]
  MoveL 500 to (274.42, 40.62, -1) mm, rotated rx -180 ry 0 rz 0 deg; joints [30.776, -53.325, 142.779, 30.777, -88.661, -0.007]
  MoveL 501 to (274.42, 142.16, -1) mm, rotated rx -180 ry 0 rz 0 deg; joints [35.47, -52.331, 138.703, 35.552, -86.177, -1.836]
  MoveL 502 to (376.02, 142.16, -1) mm, rotated rx -180 ry 0 rz 0 deg; joints [38.901, -53.92, 144.655, 38.892, -89.702, 0.734]
  MoveL 503 to (325.2, 91.37, -1) mm, rotated rx -180 ry 0 rz 0 deg; joints [34.785, -53.667, 143.9, 34.779, -89.322, 0.405]
  MoveC 504 to (324.75, 91.18, -1) mm, rotated rx 180 ry 0 rz 0 deg; joints [34.761, -53.662, 143.881, 34.755, -89.31, 0.397] to (324.3, 91.37, -1) mm, rotated rx 180 ry 0 rz 0 deg; joints [34.755, -53.654, 143.846, 34.75, -89.289, 0.382]
  MoveL 505 to (323.86, 91.82, -1) mm, rotated rx 180 ry 0 rz 0 deg; joints [34.762, -53.643, 143.801, 34.756, -89.26, 0.362]
  MoveC 506 to (323.54, 92.13, -0.81) mm, rotated rx 180 ry 0 rz 0 deg; joints [34.766, -53.653, 143.771, 34.761, -89.228, 0.34] to (323.41, 92.27, -0.37) mm, rotated rx -180 ry 0 rz 0 deg; joints [34.768, -53.691, 143.765, 34.763, -89.191, 0.314]
  Set speed (500.0 mm/s)
  MoveL 507 to (323.41, 92.27, 5) mm, rotated rx 180 ry 0 rz 0 deg; joints [34.764, -54.183, 143.84, 34.763, -88.849, 0.077]
  MoveL 508 to (302.95, 38.71, 5) mm, rotated rx -180 ry 0 rz 0 deg; joints [31.525, -54.33, 144.713, 31.519, -89.458, 0.473]
  Set speed (25.4 mm/s)
  MoveL 509 to (302.95, 38.71, 1) mm, rotated rx -180 ry 0 rz 0 deg; joints [31.528, -53.956, 144.656, 31.52, -89.727, 0.638]
  MoveL 510 to (302.95, 38.71, -0.37) mm, rotated rx 180 ry 0 rz 0 deg; joints [31.529, -53.829, 144.636, 31.521, -89.819, 0.694]
  MoveC 511 to (302.95, 38.9, -0.81) mm, rotated rx -180 ry 0 rz 0 deg; joints [31.539, -53.786, 144.623, 31.531, -89.844, 0.71] to (302.95, 39.35, -1) mm, rotated rx 180 ry 0 rz 0 deg; joints [31.561, -53.765, 144.603, 31.553, -89.844, 0.711]
  Set speed (50.8 mm/s)
  MoveL 512 to (302.95, 39.98, -1) mm, rotated rx -180 ry 0 rz 0 deg; joints [31.593, -53.76, 144.579, 31.584, -89.828, 0.701]
  MoveC 513 to (303.14, 40.43, -1) mm, rotated rx 180 ry 0 rz 0 deg; joints [31.62, -53.76, 144.574, 31.612, -89.824, 0.699] to (303.59, 40.62, -1) mm, rotated rx -180 ry 0 rz 0 deg; joints [31.643, -53.765, 144.594, 31.635, -89.837, 0.707]
  MoveL 514 to (376.02, 40.62, -1) mm, rotated rx -180 ry 0 rz 0 deg; joints [33.998, -54.649, 148.965, 34.033, -92.709, 2.687]
  MoveL 515 to (403.83, 40.62, -1) mm, rotated rx -180 ry 0 rz 0 deg; joints [34.986, -54.902, 150.59, 35.065, -93.789, 3.537]
  MoveL 516 to (403.83, 142.16, -1) mm, rotated rx -180 ry 0 rz 0 deg; joints [39.939, -54.272, 146.208, 39.932, -90.615, 1.515]
  MoveL 517 to (302.23, 40.62, -1) mm, rotated rx 180 ry 0 rz 0 deg; joints [31.602, -53.745, 144.511, 31.594, -89.782, 0.673]
  MoveL 518 to (303.59, 40.62, -1) mm, rotated rx -180 ry 0 rz 0 deg; joints [31.643, -53.765, 144.594, 31.635, -89.837, 0.707]
  MoveC 519 to (304.04, 40.43, -1) mm, rotated rx 180 ry 0 rz 0 deg; joints [31.648, -53.772, 144.629, 31.64, -89.86, 0.722] to (304.22, 39.98, -1) mm, rotated rx -180 ry 0 rz 0 deg; joints [31.631, -53.778, 144.657, 31.623, -89.879, 0.733]
  MoveL 520 to (304.22, 39.35, -1) mm, rotated rx 180 ry 0 rz 0 deg; joints [31.6, -53.783, 144.681, 31.592, -89.896, 0.743]
  MoveC 521 to (304.22, 38.9, -0.81) mm, rotated rx 180 ry 0 rz 0 deg; joints [31.577, -53.804, 144.701, 31.569, -89.895, 0.742] to (304.22, 38.71, -0.37) mm, rotated rx 180 ry 0 rz 0 deg; joints [31.568, -53.847, 144.715, 31.56, -89.87, 0.726]
  Set speed (500.0 mm/s)
  MoveL 522 to (304.22, 38.71, 5) mm, rotated rx 180 ry 0 rz 0 deg; joints [31.564, -54.348, 144.792, 31.557, -89.508, 0.504]
  MoveL 523 to (399.41, 16.27, 5) mm, rotated rx 180 ry 0 rz 0 deg; joints [33.536, -55.603, 151.391, 33.618, -93.954, 3.473]
  Set speed (25.4 mm/s)
  MoveL 524 to (399.41, 16.27, 1) mm, rotated rx -180 ry 0 rz 0 deg; joints [33.539, -55.173, 151.326, 33.636, -94.257, 3.676]
  MoveL 525 to (399.41, 16.27, -0.36) mm, rotated rx -180 ry 0 rz 0 deg; joints [33.541, -55.026, 151.303, 33.642, -94.361, 3.745]
  MoveC 526 to (399.54, 16.14, -0.81) mm, rotated rx -180 ry 0 rz 0 deg; joints [33.539, -54.98, 151.308, 33.643, -94.404, 3.774] to (399.86, 15.82, -1) mm, rotated rx -180 ry 0 rz 0 deg; joints [33.533, -54.963, 151.336, 33.639, -94.441, 3.798]
  Set speed (50.8 mm/s)
  MoveL 527 to (400.31, 15.37, -1) mm, rotated rx 180 ry 0 rz 0 deg; joints [33.525, -54.968, 151.38, 33.632, -94.474, 3.819]
  MoveC 528 to (400.49, 14.92, -1) mm, rotated rx -180 ry 0 rz 0 deg; joints [33.507, -54.971, 151.408, 33.616, -94.497, 3.831] to (400.31, 14.47, -1) mm, rotated rx -180 ry 0 rz 0 deg; joints [33.477, -54.971, 151.414, 33.585, -94.504, 3.832]
  MoveL 529 to (302.23, -83.55, -1) mm, rotated rx -180 ry 0 rz 0 deg; joints [25.056, -54.444, 148.723, 25.086, -93.007, 2.085]
  MoveL 530 to (403.83, -83.55, -1) mm, rotated rx 180 ry 0 rz 0 deg; joints [28.003, -55.114, 155.1, 28.291, -97.941, 4.987]
  MoveL 531 to (403.83, 17.99, -1) mm, rotated rx -180 ry 0 rz 0 deg; joints [33.791, -54.985, 151.484, 33.903, -94.531, 3.893]
  MoveL 532 to (400.31, 14.47, -1) mm, rotated rx -180 ry 0 rz 0 deg; joints [33.477, -54.971, 151.414, 33.585, -94.504, 3.832]
  MoveC 533 to (399.86, 14.28, -1) mm, rotated rx 180 ry 0 rz 0 deg; joints [33.451, -54.968, 151.395, 33.559, -94.492, 3.82] to (399.41, 14.47, -1) mm, rotated rx -180 ry 0 rz 0 deg; joints [33.445, -54.964, 151.362, 33.552, -94.467, 3.803]
  MoveL 534 to (398.96, 14.92, -1) mm, rotated rx 180 ry 0 rz 0 deg; joints [33.453, -54.959, 151.318, 33.558, -94.434, 3.783]
  MoveC 535 to (398.64, 15.24, -0.81) mm, rotated rx -180 ry 0 rz 0 deg; joints [33.459, -54.976, 151.29, 33.562, -94.397, 3.759] to (398.51, 15.37, -0.37) mm, rotated rx 180 ry 0 rz 0 deg; joints [33.461, -55.023, 151.285, 33.562, -94.353, 3.73]
  Set speed (500.0 mm/s)
  MoveL 536 to (398.51, 15.37, 5) mm, rotated rx -180 ry 0 rz 0 deg; joints [33.456, -55.599, 151.373, 33.538, -93.946, 3.459]
  MoveL 537 to (398.88, -106.96, 5) mm, rotated rx -180 ry 0 rz 0 deg; joints [26.412, -55.804, 155.639, 26.679, -97.933, 4.671]
  Set speed (25.4 mm/s)
  MoveL 538 to (398.88, -106.96, 1) mm, rotated rx -180 ry 0 rz 0 deg; joints [26.415, -55.327, 155.566, 26.708, -98.294, 4.855]
  MoveL 539 to (398.88, -106.96, -0.37) mm, rotated rx 180 ry 0 rz 0 deg; joints [26.416, -55.165, 155.541, 26.719, -98.416, 4.918]
  MoveC 540 to (399.01, -107.09, -0.81) mm, rotated rx -180 ry 0 rz 0 deg; joints [26.412, -55.111, 155.545, 26.719, -98.468, 4.943] to (399.33, -107.41, -1) mm, rotated rx -180 ry 0 rz 0 deg; joints [26.402, -55.089, 155.571, 26.712, -98.512, 4.963]
  Set speed (50.8 mm/s)
  MoveL 541 to (399.78, -107.86, -1) mm, rotated rx -180 ry 0 rz 0 deg; joints [26.388, -55.089, 155.612, 26.701, -98.55, 4.98]
  MoveC 542 to (399.96, -108.31, -1) mm, rotated rx 180 ry 0 rz 0 deg; joints [26.366, -55.089, 155.637, 26.68, -98.574, 4.988] to (399.78, -108.76, -1) mm, rotated rx 180 ry 0 rz 0 deg; joints [26.333, -55.088, 155.639, 26.646, -98.579, 4.984]
  MoveL 543 to (302.23, -206.24, -1) mm, rotated rx -180 ry 0 rz 0 deg; joints [17.823, -54.74, 151.873, 17.916, -95.92, 2.462]
  MoveL 544 to (403.83, -206.24, -1) mm, rotated rx -180 ry 0 rz 30 deg; joints [29.129, -54.841, 151.031, 59.194, -92.286, 5.116]
  MoveL 545 to (403.83, -104.7, -1) mm, rotated rx -180 ry 0 rz 0 deg; joints [26.709, -55.096, 155.766, 27.034, -98.654, 5.1]
  MoveL 546 to (399.78, -108.76, -1) mm, rotated rx -180 ry 0 rz 0 deg; joints [26.333, -55.088, 155.639, 26.646, -98.579, 4.984]
  MoveC 547 to (399.33, -108.94, -1) mm, rotated rx -180 ry 0 rz 0 deg; joints [26.307, -55.088, 155.617, 26.62, -98.562, 4.97] to (398.88, -108.76, -1) mm, rotated rx -180 ry 0 rz 0 deg; joints [26.305, -55.087, 155.584, 26.615, -98.533, 4.954]
  MoveL 548 to (398.43, -108.31, -1) mm, rotated rx -180 ry 0 rz 0 deg; joints [26.319, -55.087, 155.543, 26.627, -98.495, 4.938]
  MoveC 549 to (398.11, -107.99, -0.81) mm, rotated rx -180 ry 0 rz 0 deg; joints [26.329, -55.11, 155.517, 26.633, -98.451, 4.918] to (397.98, -107.86, -0.37) mm, rotated rx -180 ry 0 rz 0 deg; joints [26.333, -55.163, 155.513, 26.633, -98.4, 4.892]
  Set speed (500.0 mm/s)
  MoveL 550 to (397.98, -107.86, 5) mm, rotated rx -180 ry 0 rz 0 deg; joints [26.329, -55.802, 155.61, 26.594, -97.916, 4.647]
  MoveL 551 to (376.66, -102.8, 5) mm, rotated rx -180 ry 0 rz 0 deg; joints [25.998, -55.727, 154.128, 26.182, -96.679, 3.969]
  Set speed (25.4 mm/s)
  MoveL 552 to (376.66, -102.8, 1) mm, rotated rx 180 ry 0 rz 0 deg; joints [26.001, -55.267, 154.058, 26.205, -97.028, 4.143]
  MoveL 553 to (376.66, -102.8, -0.37) mm, rotated rx -180 ry 0 rz 0 deg; joints [26.002, -55.111, 154.034, 26.214, -97.147, 4.202]
  MoveC 554 to (376.66, -102.98, -0.81) mm, rotated rx -180 ry 0 rz 0 deg; joints [25.991, -55.06, 154.032, 26.206, -97.191, 4.222] to (376.66, -103.43, -1) mm, rotated rx -180 ry 0 rz 0 deg; joints [25.964, -55.038, 154.042, 26.18, -97.221, 4.232]
  Set speed (50.8 mm/s)
  MoveL 555 to (376.66, -104.07, -1) mm, rotated rx 180 ry 0 rz 0 deg; joints [25.926, -55.039, 154.061, 26.143, -97.241, 4.235]
  MoveC 556 to (376.47, -104.52, -1) mm, rotated rx -180 ry 0 rz 0 deg; joints [25.893, -55.038, 154.063, 26.11, -97.245, 4.231] to (376.02, -104.7, -1) mm, rotated rx 180 ry 0 rz 0 deg; joints [25.869, -55.037, 154.041, 26.084, -97.228, 4.219]
  MoveL 557 to (274.42, -104.7, -1) mm, rotated rx 180 ry 0 rz 0 deg; joints [23.179, -54.208, 147.525, 23.19, -92.18, 1.578]
  MoveL 558 to (274.42, -206.24, -1) mm, rotated rx -180 ry 0 rz 0 deg; joints [17.287, -54.511, 150.007, 17.333, -94.378, 1.908]
  MoveL 559 to (288.34, -192.34, -1) mm, rotated rx 180 ry 0 rz 0 deg; joints [18.395, -54.611, 150.643, 18.457, -94.854, 2.179]
  MoveL 560 to (376.02, -104.7, -1) mm, rotated rx 180 ry 0 rz 0 deg; joints [25.869, -55.037, 154.041, 26.084, -97.228, 4.219]
  MoveC 561 to (376.47, -104.52, -1) mm, rotated rx 180 ry 0 rz 0 deg; joints [25.893, -55.038, 154.063, 26.11, -97.245, 4.231] to (376.92, -104.7, -1) mm, rotated rx -180 ry 0 rz 0 deg; joints [25.895, -55.04, 154.097, 26.114, -97.274, 4.246]
  MoveL 562 to (377.37, -105.15, -1) mm, rotated rx -180 ry 0 rz 0 deg; joints [25.881, -55.041, 154.138, 26.102, -97.311, 4.262]
  MoveC 563 to (377.69, -105.47, -0.81) mm, rotated rx -180 ry 0 rz 0 deg; joints [25.871, -55.064, 154.171, 26.092, -97.321, 4.265] to (377.82, -105.6, -0.37) mm, rotated rx 180 ry 0 rz 0 deg; joints [25.867, -55.116, 154.191, 26.086, -97.292, 4.25]
  Set speed (500.0 mm/s)
  MoveL 564 to (377.82, -105.6, 5) mm, rotated rx -180 ry 0 rz 0 deg; joints [25.863, -55.734, 154.285, 26.053, -96.822, 4.017]
  MoveL 565 to (256.14, -102.91, 5) mm, rotated rx -180 ry 0 rz 0 deg; joints [22.845, -54.543, 146.358, 22.841, -90.803, 0.977]
  Set speed (25.4 mm/s)
  MoveL 566 to (256.14, -102.91, 1) mm, rotated rx 180 ry 0 rz 0 deg; joints [22.848, -54.158, 146.299, 22.845, -91.104, 1.104]
  MoveL 567 to (256.14, -102.91, -0.36) mm, rotated rx -180 ry 0 rz 0 deg; joints [22.849, -54.026, 146.278, 22.847, -91.206, 1.147]
  MoveC 568 to (256.27, -103.04, -0.81) mm, rotated rx -180 ry 0 rz 0 deg; joints [22.845, -53.985, 146.284, 22.843, -91.249, 1.165] to (256.59, -103.35, -1) mm, rotated rx 180 ry 0 rz 0 deg; joints [22.835, -53.973, 146.311, 22.834, -91.285, 1.18]
  Set speed (50.8 mm/s)
  MoveL 569 to (257.04, -103.8, -1) mm, rotated rx -180 ry 0 rz 0 deg; joints [22.82, -53.981, 146.353, 22.82, -91.317, 1.192]
  MoveC 570 to (257.22, -104.25, -1) mm, rotated rx -180 ry 0 rz 0 deg; joints [22.8, -53.986, 146.378, 22.8, -91.336, 1.199] to (257.04, -104.7, -1) mm, rotated rx -180 ry 0 rz 0 deg; joints [22.771, -53.985, 146.378, 22.771, -91.337, 1.198]
  MoveL 571 to (155.44, -206.24, -1) mm, rotated rx 180 ry 0 rz 0 deg; joints [15.308, -52.836, 141.787, 15.31, -88.118, -0.005]
  MoveL 572 to (257.04, -206.24, -1) mm, rotated rx -180 ry 0 rz 0 deg; joints [16.967, -54.333, 148.83, 16.992, -93.431, 1.585]
  MoveL 573 to (257.04, -104.7, -1) mm, rotated rx -180 ry 0 rz 0 deg; joints [22.771, -53.985, 146.378, 22.771, -91.337, 1.198]
  MoveC 574 to (257.22, -104.25, -1) mm, rotated rx 180 ry 0 rz 0 deg; joints [22.8, -53.986, 146.378, 22.8, -91.336, 1.199] to (257.67, -104.07, -1) mm, rotated rx 180 ry 0 rz 0 deg; joints [22.821, -53.991, 146.402, 22.82, -91.353, 1.208]
  MoveL 575 to (258.31, -104.07, -1) mm, rotated rx 180 ry 0 rz 0 deg; joints [22.835, -53.999, 146.444, 22.835, -91.384, 1.221]
  MoveC 576 to (258.76, -104.07, -0.81) mm, rotated rx 180 ry 0 rz 0 deg; joints [22.846, -54.023, 146.477, 22.846, -91.392, 1.225] to (258.94, -104.07, -0.37) mm, rotated rx 180 ry 0 rz 0 deg; joints [22.85, -54.069, 146.496, 22.85, -91.367, 1.215]
  Set speed (500.0 mm/s)
  MoveL 577 to (258.94, -104.07, 5) mm, rotated rx -180 ry 0 rz 0 deg; joints [22.846, -54.589, 146.576, 22.843, -90.962, 1.044]
  MoveL 578 to (229.86, -102.8, 5) mm, rotated rx -180 ry 0 rz 0 deg; joints [22.259, -54.144, 144.601, 22.252, -89.553, 0.445]
  Set speed (25.4 mm/s)
  MoveL 579 to (229.86, -102.8, 1) mm, rotated rx 180 ry 0 rz 0 deg; joints [22.261, -53.772, 144.544, 22.254, -89.845, 0.565]
  MoveL 580 to (229.86, -102.8, -0.37) mm, rotated rx -180 ry 0 rz 0 deg; joints [22.262, -53.645, 144.524, 22.255, -89.944, 0.605]
  MoveC 581 to (229.86, -102.98, -0.81) mm, rotated rx -180 ry 0 rz 0 deg; joints [22.252, -53.604, 144.522, 22.245, -89.98, 0.62] to (229.86, -103.43, -1) mm, rotated rx -180 ry 0 rz 0 deg; joints [22.228, -53.589, 144.532, 22.221, -90.003, 0.629]
  Set speed (50.8 mm/s)
  MoveL 582 to (229.86, -104.07, -1) mm, rotated rx 180 ry 0 rz 0 deg; joints [22.194, -53.592, 144.549, 22.187, -90.016, 0.634]
  MoveC 583 to (229.67, -104.52, -1) mm, rotated rx -180 ry 0 rz 0 deg; joints [22.166, -53.592, 144.549, 22.159, -90.017, 0.633] to (229.23, -104.7, -1) mm, rotated rx -180 ry 0 rz 0 deg; joints [22.146, -53.586, 144.524, 22.139, -89.999, 0.626]
  MoveL 584 to (127.63, -104.7, -1) mm, rotated rx 180 ry 0 rz 0 deg; joints [20.116, -51.741, 137.547, 20.183, -85.194, -1.173]
